// TwinCAT 3 PLC project PLC
// ProgramVersion: 3.1.4023.0
// libraries:
//   Tc2_Standard, * (Beckhoff Automation GmbH)
//   Tc2_System, * (Beckhoff Automation GmbH)
//   Tc3_Module, * (Beckhoff Automation GmbH)
// project tree:
//   / PlcTask.TcTTO
//   POUs/ MAIN.TcPOU
//   DUTs/IO/PDOs/ InfoData_6F19DB2B.TcDUT, Inputs_CC16D1F4.TcDUT, Outputs_D8BAB3B3.TcDUT, WcState_9091E0EB.TcDUT, InfoData_90184F0C.TcDUT, Channel_87C95E76.TcDUT, InfoData_32EB74EA.TcDUT, Channel_70C997F3.TcDUT, EPM_Inputs_Channel_385E794A.TcDUT, EMPTY_STRUCTURE.TcDUT, Device_Status_Mapping_61F79077.TcDUT, Channel_954C2EED.TcDUT, Channel_60E28ED2.TcDUT, Channel_7DE26195.TcDUT, Channel_2E0D480D.TcDUT, Channel_61FC1536.TcDUT, Channel_16463F74.TcDUT, Channel_707BD1FE.TcDUT, Channel_7D202F58.TcDUT, Channel_6CC0E226.TcDUT, Channel_0F0CD940.TcDUT, Channel_65B76600.TcDUT, Channel_72DF6336.TcDUT, Channel_22DCD695.TcDUT, Channel_3C1A6500.TcDUT, Channel_B5275D8E.TcDUT, Channel_03CEAA5E.TcDUT, Channel_1D6668A9.TcDUT, Channel_6B723A16.TcDUT, Channel_460B8C40.TcDUT, Channel_DCF170BB.TcDUT, Channel_26FC8FD8.TcDUT, Channel_FEA3DBF8.TcDUT, Channel_0D1929F0.TcDUT, Channel_6576A681.TcDUT, Channel_2589C8DC.TcDUT, Channel_BF3661CD.TcDUT, Channel_2EC3E8CA.TcDUT, Channel_F5DB8AD1.TcDUT, Channel_6D8B740B.TcDUT, Channel_2DA3FF3C.TcDUT, Channel_0514A8FA.TcDUT, Channel_4E9D1E2D.TcDUT, Channel_78571FB4.TcDUT, Channel_87905831.TcDUT, Channel_099BCCDA.TcDUT, Channel_82ADD076.TcDUT, Channel_332F026B.TcDUT, Channel_A6A8AB45.TcDUT, Channel_A42BCA5C.TcDUT, Channel_08506BCE.TcDUT, Channel_08533804.TcDUT, Channel_A04AC4BD.TcDUT, Channel_77910383.TcDUT, Channel_9BC0092E.TcDUT, Channel_7606D989.TcDUT, Channel_6931CC5B.TcDUT, Channel_F7FDEFA0.TcDUT, Channel_A1C14FB4.TcDUT, Channel_A4B48F2D.TcDUT, Channel_9E293686.TcDUT, Channel_F84AC14F.TcDUT, Channel_2F314509.TcDUT, Channel_D9D48807.TcDUT, Channel_D13646E3.TcDUT, Channel_3263D8D5.TcDUT, Channel_D490E973.TcDUT, KL_6576A681.TcDUT, Channel_64AAC8C7.TcDUT, Channel_471FAA5C.TcDUT, Diag_1F4F4573.TcDUT, Channel_0029832E.TcDUT, Channel_12652743.TcDUT, InfoData_E68C61CD.TcDUT, WcState_0B2B16F9.TcDUT, InfoData_2A97D6CF.TcDUT, Inputs_25A0042B.TcDUT, Outputs_2397A10E.TcDUT
//   DUTs/IO/Boxes/ EK1100_1FC0878B.TcDUT, EK1122_1FC0878B.TcDUT, BK1250_A2FCADE7.TcDUT, KL1002_BB38DA8F.TcDUT, BK1120_6D44499E.TcDUT, BK1120_A2FCADE7.TcDUT, CPXXXX_A2FCADE7.TcDUT, BK1150_A2FCADE7.TcDUT, IL2300_A2FCADE7.TcDUT, KL_D4CFBC22.TcDUT, KL_8EF4D3E9.TcDUT, IL2301_A2FCADE7.TcDUT, IL2302_A2FCADE7.TcDUT, CU1123_1FC0878B.TcDUT, CU1124_1FC0878B.TcDUT, CU1128_1FC0878B.TcDUT, CU1521_1FC0878B.TcDUT, CU1561_1FC0878B.TcDUT, CU2508_1FC0878B.TcDUT, CU2508_EEB2FEF4.TcDUT, CU2508_6BF2ACBC.TcDUT, CX1100_1FC0878B.TcDUT, CX5010_EtherCAT_slave_FEF7A27A.TcDUT, CX5020_EtherCAT_slave_FEF7A27A.TcDUT, CX8010_EtherCAT_slave_FEF7A27A.TcDUT, CX8110_EtherCAT_slave_FEF7A27A.TcDUT, CX2020_EtherCAT_slave_FEF7A27A.TcDUT, CX2030_EtherCAT_slave_FEF7A27A.TcDUT, CX2033_EtherCAT_slave_FEF7A27A.TcDUT, CX2040_EtherCAT_slave_FEF7A27A.TcDUT, CX2042_EtherCAT_slave_FEF7A27A.TcDUT, CX2043_EtherCAT_slave_FEF7A27A.TcDUT, CX2062_EtherCAT_slave_FEF7A27A.TcDUT, CX2072_EtherCAT_slave_FEF7A27A.TcDUT, CX9020_EtherCAT_slave_FEF7A27A.TcDUT, CX5120_EtherCAT_slave_FEF7A27A.TcDUT, CX5130_EtherCAT_slave_FEF7A27A.TcDUT, CX5140_EtherCAT_slave_FEF7A27A.TcDUT, CX5230_EtherCAT_slave_FEF7A27A.TcDUT, CX5240_EtherCAT_slave_FEF7A27A.TcDUT, KL_5E2F016F.TcDUT, KL_2EA97E3E.TcDUT, KL_1187B721.TcDUT, KL_E991A364.TcDUT, KL_063F0990.TcDUT, KL_5AE00A1C.TcDUT, KL_CFA8830D.TcDUT, KL_DBC0B844.TcDUT, KL_6930B3B2.TcDUT, KL_4F0DAD84.TcDUT, KL_2227C35B.TcDUT, KL_E653A8C1.TcDUT, KL1012_BB38DA8F.TcDUT, KL1032_BB38DA8F.TcDUT, KL1052_BB38DA8F.TcDUT, KL1104_4A257D2B.TcDUT, KL1114_4A257D2B.TcDUT, KL1124_4A257D2B.TcDUT, KL1154_4A257D2B.TcDUT, KL1164_4A257D2B.TcDUT, KL1184_4A257D2B.TcDUT, KL1194_4A257D2B.TcDUT, KL1212_EC84F46C.TcDUT, KL1232_BB38DA8F.TcDUT, KL1302_BB38DA8F.TcDUT, KL1304_4A257D2B.TcDUT, KL1312_BB38DA8F.TcDUT, KL1314_4A257D2B.TcDUT, KL1352_B54AC54D.TcDUT, KL1362_B54AC54D.TcDUT, KL1382_B54AC54D.TcDUT, KL1402_BB38DA8F.TcDUT, KL1404_4A257D2B.TcDUT, KL1408_8EF4D3E9.TcDUT, KL1412_BB38DA8F.TcDUT, KL1414_4A257D2B.TcDUT, KL1418_8EF4D3E9.TcDUT, KL1434_4A257D2B.TcDUT, KL1488_8EF4D3E9.TcDUT, KL1498_8EF4D3E9.TcDUT, KL1501_EE1D4506.TcDUT, KL_62DC61BC.TcDUT, KL1512_78388DBB.TcDUT, KL1702_BB38DA8F.TcDUT, KL1704_4A257D2B.TcDUT, KL1712_BB38DA8F.TcDUT, KL_BB38DA8F.TcDUT, KL1722_BB38DA8F.TcDUT, KL1804_4A257D2B.TcDUT, KL1808_8EF4D3E9.TcDUT, KL1809_65B88BEE.TcDUT, KL1814_4A257D2B.TcDUT, KL1819_65B88BEE.TcDUT, KL1859_C5B2A062.TcDUT, KL1862_65B88BEE.TcDUT, KL_65B88BEE.TcDUT, KL1872_65B88BEE.TcDUT, KL1889_65B88BEE.TcDUT, KL1904_7F0D69A9.TcDUT, KL1908_7F0D69A9.TcDUT, KL_ABE34026.TcDUT, KL_E882B8F1.TcDUT, KL_52751275.TcDUT, KL2012_DCA75612.TcDUT, KL2022_DCA75612.TcDUT, KL2032_DCA75612.TcDUT, KL2114_E49EE1EF.TcDUT, KL2124_E49EE1EF.TcDUT, KL2134_E49EE1EF.TcDUT, KL2184_E49EE1EF.TcDUT, KL2212_BA18203A.TcDUT, KL1202_EC84F46C.TcDUT, KL2404_E49EE1EF.TcDUT, KL2408_CBAD53BF.TcDUT, KL2424_E49EE1EF.TcDUT, KL2442_DCA75612.TcDUT, KL2488_CBAD53BF.TcDUT, KL2284_008A18FD.TcDUT, KL2502_78388DBB.TcDUT, KL2512_78388DBB.TcDUT, KL2521_D5F34107.TcDUT, KL2531_D5AE5504.TcDUT, KL_5C335388.TcDUT, KL2532_B0461874.TcDUT, KL2535_B0461874.TcDUT, KL_501418F2.TcDUT, KL2541_D5AE5504.TcDUT, KL2542_B0461874.TcDUT, KL2545_B0461874.TcDUT, KL2552_B0461874.TcDUT, KL2602_DCA75612.TcDUT, KL_DCA75612.TcDUT, KL2612_DCA75612.TcDUT, KL2622_DCA75612.TcDUT, KL2631_DE78D366.TcDUT, KL2634_E49EE1EF.TcDUT, KL2641_8487B205.TcDUT, KL_AF699C3C.TcDUT, KL2652_DCA75612.TcDUT, KL_6148C904.TcDUT, KL2701_DE78D366.TcDUT, KL2702_DCA75612.TcDUT, KL2712_DCA75612.TcDUT, KL2722_DCA75612.TcDUT, KL2732_DCA75612.TcDUT, KL2744_E49EE1EF.TcDUT, KL2751_6148C904.TcDUT, KL2761_6148C904.TcDUT, KL2784_E49EE1EF.TcDUT, KL2791_6148C904.TcDUT, KL2794_E49EE1EF.TcDUT, KL2798_CBAD53BF.TcDUT, KL2808_CBAD53BF.TcDUT, KL2819_28D63841.TcDUT, KL2828_CBAD53BF.TcDUT, KL2809_F0D0C9F8.TcDUT, KL2872_F0D0C9F8.TcDUT, KL2889_F0D0C9F8.TcDUT, KL2904_7F0D69A9.TcDUT, KL_F0D0C9F8.TcDUT, KL_CF002DCA.TcDUT, KL_F7A5EEBF.TcDUT, KL_E49EE1EF.TcDUT, KL_F206FFFF.TcDUT, KL_13ED1AE5.TcDUT, KL2774_6148C904.TcDUT, KL_CBAD53BF.TcDUT, KL3001_6148C904.TcDUT, KL3002_B0461874.TcDUT, KL3011_6148C904.TcDUT, KL3012_B0461874.TcDUT, KL3021_6148C904.TcDUT, KL3022_B0461874.TcDUT, KL3041_6148C904.TcDUT, KL3042_B0461874.TcDUT, KL3044_8BE38B75.TcDUT, KL_ACD69469.TcDUT, KL3051_6148C904.TcDUT, KL3052_B0461874.TcDUT, KL3054_8BE38B75.TcDUT, KL3061_6148C904.TcDUT, KL3062_B0461874.TcDUT, KL3064_8BE38B75.TcDUT, KL3102_B0461874.TcDUT, KL3112_B0461874.TcDUT, KL3122_B0461874.TcDUT, KL3132_B0461874.TcDUT, KL3142_78388DBB.TcDUT, KL3152_78388DBB.TcDUT, KL3158_8BE38B75.TcDUT, KL3162_78388DBB.TcDUT, KL3172_78388DBB.TcDUT, KL_78388DBB.TcDUT, KL3182_B0461874.TcDUT, KL3201_6148C904.TcDUT, KL3202_B0461874.TcDUT, KL3204_8BE38B75.TcDUT, KL_8BE38B75.TcDUT, KL3214_8BE38B75.TcDUT, KL3222_B0461874.TcDUT, KL3224_8BE38B75.TcDUT, KL3228_8BE38B75.TcDUT, KL3302_B0461874.TcDUT, KL3311_6148C904.TcDUT, KL3312_B0461874.TcDUT, KL3314_8BE38B75.TcDUT, KL3351_33637CB0.TcDUT, KL_C7B8B3CA.TcDUT, KL3356_E004D4E2.TcDUT, KL_EE1D4506.TcDUT, KL3361_73CB82BA.TcDUT, KL_73CB82BA.TcDUT, KL3362_E98BF8F1.TcDUT, KL6211_60136EA1.TcDUT, KL_9AE543B6.TcDUT, KL_FC0201B8.TcDUT, KL_498D8863.TcDUT, KL_71341691.TcDUT, KL_2B11657C.TcDUT, KL6224_C0F107BD.TcDUT, KL_FC1E3393.TcDUT, KL_C51B1CB0.TcDUT, KL_7EC2CD64.TcDUT, KL_3829421A.TcDUT, KL_9116C2C1.TcDUT, KL6551_528AE398.TcDUT, KL_3325E583.TcDUT, KL_528AE398.TcDUT, KL6781_BE595CA2.TcDUT, KL6811_6148C904.TcDUT, KL6821_F77C82D2.TcDUT, KL6831_BE595CA2.TcDUT, KL6841_BE595CA2.TcDUT, KL6904_B938D612.TcDUT, KL_921B772D.TcDUT, KL_779990DF.TcDUT, KL8001_7761653A.TcDUT, KL8519_8C34650F.TcDUT, KL8524_A4B9216E.TcDUT, KL8528_73A97EC1.TcDUT, KL8548_23451728.TcDUT, KL8610_C571D068.TcDUT, KL_5A83E84C.TcDUT, KL_BF4AA06C.TcDUT, KL_7485E925.TcDUT, KL_372C6BEC.TcDUT, KL_2E5CD6C8.TcDUT, KL_68BDE1E9.TcDUT, KL_84AAE8B6.TcDUT, KL9110_8BEE55F2.TcDUT, KL9160_8BEE55F2.TcDUT, KL9191_962A24DF.TcDUT, KL9210_8BEE55F2.TcDUT, KL9260_8BEE55F2.TcDUT, KL_E4BD2B38.TcDUT, KL9528_8C984603.TcDUT, KL9999_7A10A7F6.TcDUT
//   DUTs/IO/Devices/ SyncUnitTask_2D604ED5.TcDUT, SyncUnitTasks_6FEB8257.TcDUT, SyncUnits_99E584AF.TcDUT
//   DUTs/IO/Topology/ A_0014_BK1250_0000_0000_09E1EB45.TcDUT, Beckhoff_BKxxxxsub_EK1100_59A46924.TcDUT, A_0001_BK1120_0000_0000_205E6559.TcDUT, A_0002_BK1120_0000_0001_76F1F8EB.TcDUT, A_0003_BK1120_0000_0016_8D015E3D.TcDUT, A_0004_BK1120_0000_0017_DBAEC38F.TcDUT, A_0005_BK1120_0000_0018_C2DFD8D8.TcDUT, A_0006_BK1120_0000_0019_9470456A.TcDUT, A_0007_BK1120_0000_0020_61E27259.TcDUT, A_0008_BK1120_0000_0021_374DEFEB.TcDUT, A_0009_CPXXXX_BK1150_0016_CCBD493D.TcDUT, A_0010_BK1150_0000_0016_9A12D48F.TcDUT, A_0011_BK1150_0000_0017_3F9D1926.TcDUT, A_0012_BK1150_0000_0018_69328494.TcDUT, A_0013_BK1150_0000_0019_92C22242.TcDUT, A_0016_BK1250_0000_0017_C46DBFF0.TcDUT, Term_19_EK1100_718FBBA4.TcDUT, A_0018_BK1250_0000_0019_DD1CA4A7.TcDUT, Term_23_EK1100_08A82DAA.TcDUT, A_0017_BK1250_0000_0018_8BB33915.TcDUT, Term_21_EK1100_FD75FF18.TcDUT, A_0019_IL2300_B110_0016_AC908CDE.TcDUT, A_0020_IL2300_B110_0017_8C062E24.TcDUT, A_0021_IL2301_B110_0016_FF61810D.TcDUT, A_0022_IL2301_B110_0017_BAC34F2E.TcDUT, A_0023_IL2302_B110_0016_19AEDF5F.TcDUT, A_0024_IL2302_B110_0017_E18CEC30.TcDUT, Beckhoff_BKxxxxEK1122_C32C6A5C.TcDUT, A_0015_BK1250_0000_0016_5F4E76F7.TcDUT, Beckhoff_BKxxxx_735133AB.TcDUT, A_0006_CU1128_0000_0002_093CCA2E.TcDUT, A_0005_CU1128_0000_0001_8DEFD527.TcDUT, A_0004_CU1128_0000_0000_2F60DA9F.TcDUT, A_0003_CU1124_0000_0016_CE6B0448.TcDUT, A_0002_CU1123_0010_0016_E68B3D99.TcDUT, A_0001_CU1123_0000_0016_30E128CC.TcDUT, Beckhoff_CUxxxxEK1122_BE344318.TcDUT, Beckhoff_CUxxxx_E9AD9532.TcDUT, Beckhoff_CXxxxxEK1122_ADC91C0D.TcDUT, Beckhoff_CXxxxx_7C0A3C1E.TcDUT, TcTerminals210_1BK1250_A7ABB5AA.TcDUT, TcTerminals210_EK1100_1_5C778379.TcDUT, TcTerminals210_2BK1250_CEF74155.TcDUT, TcTerminals210_EK1100_2_50C14331.TcDUT, EtherCAT_Master_BKCUCX_25A199DC.TcDUT
//   DUTs/IO/Base/ EtcSlaveBase_82538BE2.TcDUT, EtcSlaveBase_82538BE2.TcDUT, EtcSlaveBase_82538BE2.TcDUT, EtcSlaveTerminalBase_947E5A46.TcDUT, EtcSlaveBoxBase_77A0E4A7.TcDUT, EtcSlaveEndTerminalBase_866C7F0C.TcDUT, InputBase_8311D824.TcDUT, OutputBase_10CEE7DE.TcDUT, EtcMasterBase_62654B43.TcDUT
//   GVLs/ GVL_iXlinker.TcGVL
// real-time tasks:
//   TASK PlcTask: cycle T#10ms, priority 20, ADS port 350
// I/O:
//   DEVICE EtherCAT_Master_BKCUCX, AmsNetId 172.20.30.238.6.1
//     Beckhoff BKxxxx [EK1100 EtherCAT Coupler (2A E-Bus)]
//       Beckhoff BKxxxxEK1122 [EK1122 2 port EtherCAT junction]
//         Beckhoff BKxxxxsub EK1100 [EK1100 EtherCAT Coupler (2A E-Bus)]
//           A_0014(BK1250-0000-0000)
//         A_0001(BK1120-0000-0000)
//         A_0002(BK1120-0000-0001)
//         A_0003(BK1120-0000-0016)
//         A_0004(BK1120-0000-0017)
//         A_0005(BK1120-0000-0018)
//         A_0006(BK1120-0000-0019)
//         A_0007(BK1120-0000-0020)
//         A_0008(BK1120-0000-0021)
//         A_0009(CPXXXX-BK1150-0016)
//         A_0010(BK1150-0000-0016)
//         A_0011(BK1150-0000-0017)
//         A_0012(BK1150-0000-0018)
//         A_0013(BK1150-0000-0019)
//         Term 19 (EK1100) [EK1100 EtherCAT Coupler (2A E-Bus)]
//           A_0016(BK1250-0000-0017)
//         Term 23 (EK1100) [EK1100 EtherCAT Coupler (2A E-Bus)]
//           A_0018(BK1250-0000-0019)
//         Term 21 (EK1100) [EK1100 EtherCAT Coupler (2A E-Bus)]
//           A_0017(BK1250-0000-0018)
//         A_0019(IL2300-B110-0016)
//         A_0020(IL2300-B110-0017)
//         A_0021(IL2301-B110-0016)
//         A_0022(IL2301-B110-0017)
//         A_0023(IL2302-B110-0016)
//         A_0024(IL2302-B110-0017)
//       A_0015(BK1250-0000-0016)
//     Beckhoff CUxxxx [EK1100 EtherCAT Coupler (2A E-Bus)]
//       Beckhoff CUxxxxEK1122 [EK1122 2 port EtherCAT junction]
//         Beckhoff CUxxxxsub EK1100 [EK1100 EtherCAT Coupler (2A E-Bus)]
//         A_0001(CU1123-0000-0016) [CU1123 EtherCAT junction (3-ports)]
//           A_0002(CU1123-0010-0016) [CU1123-0010 EtherCAT junction (3-ports, Extended Distance)]
//             A_0003(CU1124-0000-0016) [CU1124 EtherCAT junction (4-ports)]
//               A_0004(CU1128-0000-0000) [CU1128 6x EtherCAT junction]
//                 A_0005(CU1128-0000-0001) [CU1128 6x EtherCAT junction]
//                   A_0006(CU1128-0000-0002) [CU1128 6x EtherCAT junction]
//                     A_0007(CU1521-0010-0000) [CU1521-0010 EtherCAT media converter (Singlemode)]
//                     A_0008(CU1561-0000-0000) [CU1561 EtherCAT media converter (POF)]
//                     A_0009(CU2508-0000-0000) [CU2508 Ethernet Port]
//                     A_0010(CU2508-0000-0016) [CU2508 Configuration Port]
//                     A_0011(CU2508-0000-0017) [CU2508 Configuration Port]
//                     A_0012(CU2508-0000-0018) [CU2508 Configuration Port]
//                     A_0013(CU2508-0000-0019) [CU2508 Configuration Port]
//                     A_0006(CU1128-0000-0002)_2 (CU1128-B) [CU1128 6x EtherCAT junction - Dev A]
//                     A_0006(CU1128-0000-0002)_3 (CU1128-C) [CU1128 6x EtherCAT junction - Dev B]
//                   A_0005(CU1128-0000-0001)_2 (CU1128-B) [CU1128 6x EtherCAT junction - Dev A]
//                   A_0005(CU1128-0000-0001)_3 (CU1128-C) [CU1128 6x EtherCAT junction - Dev B]
//                 A_0004(CU1128-0000-0000)_2 (CU1128-B) [CU1128 6x EtherCAT junction - Dev A]
//                 A_0004(CU1128-0000-0000)_3 (CU1128-C) [CU1128 6x EtherCAT junction - Dev B]
//     Beckhoff CXxxxx [EK1100 EtherCAT Coupler (2A E-Bus)]
//       Beckhoff CXxxxxEK1122 [EK1122 2 port EtherCAT junction]
//         Beckhoff CXxxxxsub EK1100 [EK1100 EtherCAT Coupler (2A E-Bus)]
//         A_0001(CX1100-0004-0000) [CX1100-0004 EtherCAT Power supply (2A E-Bus)]
//         A_0003(CX1100-0004-0002) [CX1100-0004 EtherCAT Power supply (2A E-Bus)]
//         A_0004 (CX5010 EtherCAT slave) [CX5010 EtherCAT slave]
//         A_0005 (CX5010 EtherCAT slave) [CX5010 EtherCAT slave]
//         A_0006 (CX5020 EtherCAT slave) [CX5020 EtherCAT slave]
//         A_0007 (CX5020 EtherCAT slave) [CX5020 EtherCAT slave]
//         A_0008 (CX8010 EtherCAT slave) [CX8010 EtherCAT slave]
//         A_0009 (CX8010 EtherCAT slave) [CX8010 EtherCAT slave]
//         A_0010 (CX8110 EtherCAT slave) [CX8110 EtherCAT slave]
//         A_0011 (CX2020 EtherCAT slave) [CX2020 EtherCAT slave]
//         A_0012 (CX2020 EtherCAT slave) [CX2020 EtherCAT slave]
//         A_0013 (CX2020 EtherCAT slave) [CX2020 EtherCAT slave]
//         A_0014 (CX2030 EtherCAT slave) [CX2030 EtherCAT slave]
//         A_0015 (CX2030 EtherCAT slave) [CX2030 EtherCAT slave]
//         A_0016 (CX2030 EtherCAT slave) [CX2030 EtherCAT slave]
//         A_0017 (CX2033 EtherCAT slave) [CX2033 EtherCAT slave]
//         A_0018 (CX2040 EtherCAT slave) [CX2040 EtherCAT slave]
//         A_0019 (CX2040 EtherCAT slave) [CX2040 EtherCAT slave]
//         A_0020 (CX2040 EtherCAT slave) [CX2040 EtherCAT slave]
//         A_0021 (CX2042 EtherCAT slave) [CX2042 EtherCAT slave]
//         A_0022 (CX2043 EtherCAT slave) [CX2043 EtherCAT slave]
//         A_0023 (CX2062 EtherCAT slave) [CX2062 EtherCAT slave]
//         A_0024 (CX2072 EtherCAT slave) [CX2072 EtherCAT slave]
//         A_0025 (CX9020 EtherCAT slave) [CX9020 EtherCAT slave]
//         A_0026 (CX9020 EtherCAT slave) [CX9020 EtherCAT slave]
//         A_0027 (CX5120 EtherCAT slave) [CX5120 EtherCAT slave]
//         A_0028 (CX5130 EtherCAT slave) [CX5130 EtherCAT slave]
//         A_0029 (CX5140 EtherCAT slave) [CX5140 EtherCAT slave]
//         A_0030 (CX5230 EtherCAT slave) [CX5230 EtherCAT slave]
//         A_0031 (CX5240 EtherCAT slave) [CX5240 EtherCAT slave]
//         A_0002(CX1100-0004-0001) [CX1100-0004 EtherCAT Power supply (2A E-Bus)]
//     TcTerminals210_EK1100_1 [EK1100 EtherCAT Coupler (2A E-Bus)]
//       TcTerminals210_1BK1250
//     TcTerminals210_EK1100_2 [EK1100 EtherCAT Coupler (2A E-Bus)]
//       TcTerminals210_2BK1250
// variable links:
//   PLC/PLC Instance <-> EtherCAT Master BKCUCX/Beckhoff BKxxxx
//     PlcTask Inputs/GVL_iXlinker.EtherCAT_Master_BKCUCX.Beckhoff_BKxxxx.InfoData.State <-> InfoData/State
//   PLC/PLC Instance <-> EtherCAT Master BKCUCX/Beckhoff BKxxxx/Beckhoff BKxxxxEK1122
//     PlcTask Inputs/GVL_iXlinker.EtherCAT_Master_BKCUCX.Beckhoff_BKxxxx.Beckhoff_BKxxxxEK1122.InfoData.State <-> InfoData/State
//   PLC/PLC Instance <-> EtherCAT Master BKCUCX/Beckhoff BKxxxx/Beckhoff BKxxxxEK1122/Beckhoff BKxxxxsub EK1100
//     PlcTask Inputs/GVL_iXlinker.EtherCAT_Master_BKCUCX.Beckhoff_BKxxxx.Beckhoff_BKxxxxEK1122.Beckhoff_BKxxxxsub_EK1100.InfoData.State <-> InfoData/State
//   PLC/PLC Instance <-> EtherCAT Master BKCUCX/Beckhoff BKxxxx/Beckhoff BKxxxxEK1122/Beckhoff BKxxxxsub EK1100/A_0014(BK1250-0000-0000)
//     PlcTask Inputs/GVL_iXlinker.EtherCAT_Master_BKCUCX.Beckhoff_BKxxxx.Beckhoff_BKxxxxEK1122.Beckhoff_BKxxxxsub_EK1100.A_0014_BK1250_0000_0000.Inputs.CouplerState <-> Inputs/CouplerState
//     PlcTask Inputs/GVL_iXlinker.EtherCAT_Master_BKCUCX.Beckhoff_BKxxxx.Beckhoff_BKxxxxEK1122.Beckhoff_BKxxxxsub_EK1100.A_0014_BK1250_0000_0000.Outputs.CouplerCtrl <-> Outputs/CouplerCtrl
//     PlcTask Inputs/GVL_iXlinker.EtherCAT_Master_BKCUCX.Beckhoff_BKxxxx.Beckhoff_BKxxxxEK1122.Beckhoff_BKxxxxsub_EK1100.A_0014_BK1250_0000_0000.WcState.WcState <-> WcState/WcState
//     PlcTask Inputs/GVL_iXlinker.EtherCAT_Master_BKCUCX.Beckhoff_BKxxxx.Beckhoff_BKxxxxEK1122.Beckhoff_BKxxxxsub_EK1100.A_0014_BK1250_0000_0000.WcState.InputToggle <-> WcState/InputToggle
//     PlcTask Inputs/GVL_iXlinker.EtherCAT_Master_BKCUCX.Beckhoff_BKxxxx.Beckhoff_BKxxxxEK1122.Beckhoff_BKxxxxsub_EK1100.A_0014_BK1250_0000_0000.InfoData.AdsAddr <-> InfoData/AdsAddr
//     PlcTask Inputs/GVL_iXlinker.EtherCAT_Master_BKCUCX.Beckhoff_BKxxxx.Beckhoff_BKxxxxEK1122.Beckhoff_BKxxxxsub_EK1100.A_0014_BK1250_0000_0000.InfoData.AoeNetId <-> InfoData/AoeNetId
//     PlcTask Inputs/GVL_iXlinker.EtherCAT_Master_BKCUCX.Beckhoff_BKxxxx.Beckhoff_BKxxxxEK1122.Beckhoff_BKxxxxsub_EK1100.A_0014_BK1250_0000_0000.InfoData.State <-> InfoData/State
//   PLC/PLC Instance <-> EtherCAT Master BKCUCX/Beckhoff BKxxxx/Beckhoff BKxxxxEK1122/Beckhoff BKxxxxsub EK1100/A_0014(BK1250-0000-0000)/Term 397 (KL1002)
//     PlcTask Inputs/GVL_iXlinker.EtherCAT_Master_BKCUCX.Beckhoff_BKxxxx.Beckhoff_BKxxxxEK1122.Beckhoff_BKxxxxsub_EK1100.A_0014_BK1250_0000_0000.Term_397_KL1002.Channel_1.Input <-> Channel 1/Input
//     PlcTask Inputs/GVL_iXlinker.EtherCAT_Master_BKCUCX.Beckhoff_BKxxxx.Beckhoff_BKxxxxEK1122.Beckhoff_BKxxxxsub_EK1100.A_0014_BK1250_0000_0000.Term_397_KL1002.Channel_2.Input <-> Channel 2/Input
//   PLC/PLC Instance <-> EtherCAT Master BKCUCX/Beckhoff BKxxxx/Beckhoff BKxxxxEK1122/A_0001(BK1120-0000-0000)
//     PlcTask Inputs/GVL_iXlinker.EtherCAT_Master_BKCUCX.Beckhoff_BKxxxx.Beckhoff_BKxxxxEK1122.A_0001_BK1120_0000_0000.Inputs.CouplerState <-> Inputs/CouplerState
//     PlcTask Inputs/GVL_iXlinker.EtherCAT_Master_BKCUCX.Beckhoff_BKxxxx.Beckhoff_BKxxxxEK1122.A_0001_BK1120_0000_0000.Outputs.CouplerCtrl <-> Outputs/CouplerCtrl
//     PlcTask Inputs/GVL_iXlinker.EtherCAT_Master_BKCUCX.Beckhoff_BKxxxx.Beckhoff_BKxxxxEK1122.A_0001_BK1120_0000_0000.WcState.WcState <-> WcState/WcState
//     PlcTask Inputs/GVL_iXlinker.EtherCAT_Master_BKCUCX.Beckhoff_BKxxxx.Beckhoff_BKxxxxEK1122.A_0001_BK1120_0000_0000.WcState.InputToggle <-> WcState/InputToggle
//     PlcTask Inputs/GVL_iXlinker.EtherCAT_Master_BKCUCX.Beckhoff_BKxxxx.Beckhoff_BKxxxxEK1122.A_0001_BK1120_0000_0000.InfoData.AdsAddr <-> InfoData/AdsAddr
//     PlcTask Inputs/GVL_iXlinker.EtherCAT_Master_BKCUCX.Beckhoff_BKxxxx.Beckhoff_BKxxxxEK1122.A_0001_BK1120_0000_0000.InfoData.State <-> InfoData/State
//   PLC/PLC Instance <-> EtherCAT Master BKCUCX/Beckhoff BKxxxx/Beckhoff BKxxxxEK1122/A_0001(BK1120-0000-0000)/Term 374 (KL1002)
//     PlcTask Inputs/GVL_iXlinker.EtherCAT_Master_BKCUCX.Beckhoff_BKxxxx.Beckhoff_BKxxxxEK1122.A_0001_BK1120_0000_0000.Term_374_KL1002.Channel_1.Input <-> Channel 1/Input
//     PlcTask Inputs/GVL_iXlinker.EtherCAT_Master_BKCUCX.Beckhoff_BKxxxx.Beckhoff_BKxxxxEK1122.A_0001_BK1120_0000_0000.Term_374_KL1002.Channel_2.Input <-> Channel 2/Input
//   PLC/PLC Instance <-> EtherCAT Master BKCUCX/Beckhoff BKxxxx/Beckhoff BKxxxxEK1122/A_0002(BK1120-0000-0001)
//     PlcTask Inputs/GVL_iXlinker.EtherCAT_Master_BKCUCX.Beckhoff_BKxxxx.Beckhoff_BKxxxxEK1122.A_0002_BK1120_0000_0001.Inputs.CouplerState <-> Inputs/CouplerState
//     PlcTask Inputs/GVL_iXlinker.EtherCAT_Master_BKCUCX.Beckhoff_BKxxxx.Beckhoff_BKxxxxEK1122.A_0002_BK1120_0000_0001.Outputs.CouplerCtrl <-> Outputs/CouplerCtrl
//     PlcTask Inputs/GVL_iXlinker.EtherCAT_Master_BKCUCX.Beckhoff_BKxxxx.Beckhoff_BKxxxxEK1122.A_0002_BK1120_0000_0001.WcState.WcState <-> WcState/WcState
//     PlcTask Inputs/GVL_iXlinker.EtherCAT_Master_BKCUCX.Beckhoff_BKxxxx.Beckhoff_BKxxxxEK1122.A_0002_BK1120_0000_0001.WcState.InputToggle <-> WcState/InputToggle
//     PlcTask Inputs/GVL_iXlinker.EtherCAT_Master_BKCUCX.Beckhoff_BKxxxx.Beckhoff_BKxxxxEK1122.A_0002_BK1120_0000_0001.InfoData.AdsAddr <-> InfoData/AdsAddr
//     PlcTask Inputs/GVL_iXlinker.EtherCAT_Master_BKCUCX.Beckhoff_BKxxxx.Beckhoff_BKxxxxEK1122.A_0002_BK1120_0000_0001.InfoData.AoeNetId <-> InfoData/AoeNetId
//     PlcTask Inputs/GVL_iXlinker.EtherCAT_Master_BKCUCX.Beckhoff_BKxxxx.Beckhoff_BKxxxxEK1122.A_0002_BK1120_0000_0001.InfoData.State <-> InfoData/State
//   PLC/PLC Instance <-> EtherCAT Master BKCUCX/Beckhoff BKxxxx/Beckhoff BKxxxxEK1122/A_0002(BK1120-0000-0001)/Term 375 (KL1002)
//     PlcTask Inputs/GVL_iXlinker.EtherCAT_Master_BKCUCX.Beckhoff_BKxxxx.Beckhoff_BKxxxxEK1122.A_0002_BK1120_0000_0001.Term_375_KL1002.Channel_1.Input <-> Channel 1/Input
//     PlcTask Inputs/GVL_iXlinker.EtherCAT_Master_BKCUCX.Beckhoff_BKxxxx.Beckhoff_BKxxxxEK1122.A_0002_BK1120_0000_0001.Term_375_KL1002.Channel_2.Input <-> Channel 2/Input
//   PLC/PLC Instance <-> EtherCAT Master BKCUCX/Beckhoff BKxxxx/Beckhoff BKxxxxEK1122/A_0003(BK1120-0000-0016)
//     PlcTask Inputs/GVL_iXlinker.EtherCAT_Master_BKCUCX.Beckhoff_BKxxxx.Beckhoff_BKxxxxEK1122.A_0003_BK1120_0000_0016.Inputs.CouplerState <-> Inputs/CouplerState
//     PlcTask Inputs/GVL_iXlinker.EtherCAT_Master_BKCUCX.Beckhoff_BKxxxx.Beckhoff_BKxxxxEK1122.A_0003_BK1120_0000_0016.Outputs.CouplerCtrl <-> Outputs/CouplerCtrl
//     PlcTask Inputs/GVL_iXlinker.EtherCAT_Master_BKCUCX.Beckhoff_BKxxxx.Beckhoff_BKxxxxEK1122.A_0003_BK1120_0000_0016.WcState.WcState <-> WcState/WcState
//     PlcTask Inputs/GVL_iXlinker.EtherCAT_Master_BKCUCX.Beckhoff_BKxxxx.Beckhoff_BKxxxxEK1122.A_0003_BK1120_0000_0016.WcState.InputToggle <-> WcState/InputToggle
//     PlcTask Inputs/GVL_iXlinker.EtherCAT_Master_BKCUCX.Beckhoff_BKxxxx.Beckhoff_BKxxxxEK1122.A_0003_BK1120_0000_0016.InfoData.AdsAddr <-> InfoData/AdsAddr
//     PlcTask Inputs/GVL_iXlinker.EtherCAT_Master_BKCUCX.Beckhoff_BKxxxx.Beckhoff_BKxxxxEK1122.A_0003_BK1120_0000_0016.InfoData.AoeNetId <-> InfoData/AoeNetId
//     PlcTask Inputs/GVL_iXlinker.EtherCAT_Master_BKCUCX.Beckhoff_BKxxxx.Beckhoff_BKxxxxEK1122.A_0003_BK1120_0000_0016.InfoData.State <-> InfoData/State
//   PLC/PLC Instance <-> EtherCAT Master BKCUCX/Beckhoff BKxxxx/Beckhoff BKxxxxEK1122/A_0003(BK1120-0000-0016)/Term 376 (KL1002)
//     PlcTask Inputs/GVL_iXlinker.EtherCAT_Master_BKCUCX.Beckhoff_BKxxxx.Beckhoff_BKxxxxEK1122.A_0003_BK1120_0000_0016.Term_376_KL1002.Channel_1.Input <-> Channel 1/Input
//     PlcTask Inputs/GVL_iXlinker.EtherCAT_Master_BKCUCX.Beckhoff_BKxxxx.Beckhoff_BKxxxxEK1122.A_0003_BK1120_0000_0016.Term_376_KL1002.Channel_2.Input <-> Channel 2/Input
//   PLC/PLC Instance <-> EtherCAT Master BKCUCX/Beckhoff BKxxxx/Beckhoff BKxxxxEK1122/A_0004(BK1120-0000-0017)
//     PlcTask Inputs/GVL_iXlinker.EtherCAT_Master_BKCUCX.Beckhoff_BKxxxx.Beckhoff_BKxxxxEK1122.A_0004_BK1120_0000_0017.Inputs.CouplerState <-> Inputs/CouplerState
//     PlcTask Inputs/GVL_iXlinker.EtherCAT_Master_BKCUCX.Beckhoff_BKxxxx.Beckhoff_BKxxxxEK1122.A_0004_BK1120_0000_0017.Outputs.CouplerCtrl <-> Outputs/CouplerCtrl
//     PlcTask Inputs/GVL_iXlinker.EtherCAT_Master_BKCUCX.Beckhoff_BKxxxx.Beckhoff_BKxxxxEK1122.A_0004_BK1120_0000_0017.WcState.WcState <-> WcState/WcState
//     PlcTask Inputs/GVL_iXlinker.EtherCAT_Master_BKCUCX.Beckhoff_BKxxxx.Beckhoff_BKxxxxEK1122.A_0004_BK1120_0000_0017.WcState.InputToggle <-> WcState/InputToggle
//     PlcTask Inputs/GVL_iXlinker.EtherCAT_Master_BKCUCX.Beckhoff_BKxxxx.Beckhoff_BKxxxxEK1122.A_0004_BK1120_0000_0017.InfoData.AdsAddr <-> InfoData/AdsAddr
//     PlcTask Inputs/GVL_iXlinker.EtherCAT_Master_BKCUCX.Beckhoff_BKxxxx.Beckhoff_BKxxxxEK1122.A_0004_BK1120_0000_0017.InfoData.AoeNetId <-> InfoData/AoeNetId
//     PlcTask Inputs/GVL_iXlinker.EtherCAT_Master_BKCUCX.Beckhoff_BKxxxx.Beckhoff_BKxxxxEK1122.A_0004_BK1120_0000_0017.InfoData.State <-> InfoData/State
//   PLC/PLC Instance <-> EtherCAT Master BKCUCX/Beckhoff BKxxxx/Beckhoff BKxxxxEK1122/A_0004(BK1120-0000-0017)/Term 377 (KL1002)
//     PlcTask Inputs/GVL_iXlinker.EtherCAT_Master_BKCUCX.Beckhoff_BKxxxx.Beckhoff_BKxxxxEK1122.A_0004_BK1120_0000_0017.Term_377_KL1002.Channel_1.Input <-> Channel 1/Input
//     PlcTask Inputs/GVL_iXlinker.EtherCAT_Master_BKCUCX.Beckhoff_BKxxxx.Beckhoff_BKxxxxEK1122.A_0004_BK1120_0000_0017.Term_377_KL1002.Channel_2.Input <-> Channel 2/Input
//   PLC/PLC Instance <-> EtherCAT Master BKCUCX/Beckhoff BKxxxx/Beckhoff BKxxxxEK1122/A_0005(BK1120-0000-0018)
//     PlcTask Inputs/GVL_iXlinker.EtherCAT_Master_BKCUCX.Beckhoff_BKxxxx.Beckhoff_BKxxxxEK1122.A_0005_BK1120_0000_0018.Inputs.CouplerState <-> Inputs/CouplerState
//     PlcTask Inputs/GVL_iXlinker.EtherCAT_Master_BKCUCX.Beckhoff_BKxxxx.Beckhoff_BKxxxxEK1122.A_0005_BK1120_0000_0018.Outputs.CouplerCtrl <-> Outputs/CouplerCtrl
//     PlcTask Inputs/GVL_iXlinker.EtherCAT_Master_BKCUCX.Beckhoff_BKxxxx.Beckhoff_BKxxxxEK1122.A_0005_BK1120_0000_0018.WcState.WcState <-> WcState/WcState
//     PlcTask Inputs/GVL_iXlinker.EtherCAT_Master_BKCUCX.Beckhoff_BKxxxx.Beckhoff_BKxxxxEK1122.A_0005_BK1120_0000_0018.WcState.InputToggle <-> WcState/InputToggle
//     PlcTask Inputs/GVL_iXlinker.EtherCAT_Master_BKCUCX.Beckhoff_BKxxxx.Beckhoff_BKxxxxEK1122.A_0005_BK1120_0000_0018.InfoData.AdsAddr <-> InfoData/AdsAddr
//     PlcTask Inputs/GVL_iXlinker.EtherCAT_Master_BKCUCX.Beckhoff_BKxxxx.Beckhoff_BKxxxxEK1122.A_0005_BK1120_0000_0018.InfoData.AoeNetId <-> InfoData/AoeNetId
//     PlcTask Inputs/GVL_iXlinker.EtherCAT_Master_BKCUCX.Beckhoff_BKxxxx.Beckhoff_BKxxxxEK1122.A_0005_BK1120_0000_0018.InfoData.State <-> InfoData/State
//   PLC/PLC Instance <-> EtherCAT Master BKCUCX/Beckhoff BKxxxx/Beckhoff BKxxxxEK1122/A_0005(BK1120-0000-0018)/Term 378 (KL1002)
//     PlcTask Inputs/GVL_iXlinker.EtherCAT_Master_BKCUCX.Beckhoff_BKxxxx.Beckhoff_BKxxxxEK1122.A_0005_BK1120_0000_0018.Term_378_KL1002.Channel_1.Input <-> Channel 1/Input
//     PlcTask Inputs/GVL_iXlinker.EtherCAT_Master_BKCUCX.Beckhoff_BKxxxx.Beckhoff_BKxxxxEK1122.A_0005_BK1120_0000_0018.Term_378_KL1002.Channel_2.Input <-> Channel 2/Input
//   PLC/PLC Instance <-> EtherCAT Master BKCUCX/Beckhoff BKxxxx/Beckhoff BKxxxxEK1122/A_0006(BK1120-0000-0019)
//     PlcTask Inputs/GVL_iXlinker.EtherCAT_Master_BKCUCX.Beckhoff_BKxxxx.Beckhoff_BKxxxxEK1122.A_0006_BK1120_0000_0019.Inputs.CouplerState <-> Inputs/CouplerState
//     PlcTask Inputs/GVL_iXlinker.EtherCAT_Master_BKCUCX.Beckhoff_BKxxxx.Beckhoff_BKxxxxEK1122.A_0006_BK1120_0000_0019.Outputs.CouplerCtrl <-> Outputs/CouplerCtrl
//     PlcTask Inputs/GVL_iXlinker.EtherCAT_Master_BKCUCX.Beckhoff_BKxxxx.Beckhoff_BKxxxxEK1122.A_0006_BK1120_0000_0019.WcState.WcState <-> WcState/WcState
//     PlcTask Inputs/GVL_iXlinker.EtherCAT_Master_BKCUCX.Beckhoff_BKxxxx.Beckhoff_BKxxxxEK1122.A_0006_BK1120_0000_0019.WcState.InputToggle <-> WcState/InputToggle
//     PlcTask Inputs/GVL_iXlinker.EtherCAT_Master_BKCUCX.Beckhoff_BKxxxx.Beckhoff_BKxxxxEK1122.A_0006_BK1120_0000_0019.InfoData.AdsAddr <-> InfoData/AdsAddr
//     PlcTask Inputs/GVL_iXlinker.EtherCAT_Master_BKCUCX.Beckhoff_BKxxxx.Beckhoff_BKxxxxEK1122.A_0006_BK1120_0000_0019.InfoData.AoeNetId <-> InfoData/AoeNetId
//     PlcTask Inputs/GVL_iXlinker.EtherCAT_Master_BKCUCX.Beckhoff_BKxxxx.Beckhoff_BKxxxxEK1122.A_0006_BK1120_0000_0019.InfoData.State <-> InfoData/State
//   PLC/PLC Instance <-> EtherCAT Master BKCUCX/Beckhoff BKxxxx/Beckhoff BKxxxxEK1122/A_0006(BK1120-0000-0019)/Term 379 (KL1002)
//     PlcTask Inputs/GVL_iXlinker.EtherCAT_Master_BKCUCX.Beckhoff_BKxxxx.Beckhoff_BKxxxxEK1122.A_0006_BK1120_0000_0019.Term_379_KL1002.Channel_1.Input <-> Channel 1/Input
//     PlcTask Inputs/GVL_iXlinker.EtherCAT_Master_BKCUCX.Beckhoff_BKxxxx.Beckhoff_BKxxxxEK1122.A_0006_BK1120_0000_0019.Term_379_KL1002.Channel_2.Input <-> Channel 2/Input
//   PLC/PLC Instance <-> EtherCAT Master BKCUCX/Beckhoff BKxxxx/Beckhoff BKxxxxEK1122/A_0007(BK1120-0000-0020)
//     PlcTask Inputs/GVL_iXlinker.EtherCAT_Master_BKCUCX.Beckhoff_BKxxxx.Beckhoff_BKxxxxEK1122.A_0007_BK1120_0000_0020.Inputs.CouplerState <-> Inputs/CouplerState
//     PlcTask Inputs/GVL_iXlinker.EtherCAT_Master_BKCUCX.Beckhoff_BKxxxx.Beckhoff_BKxxxxEK1122.A_0007_BK1120_0000_0020.Outputs.CouplerCtrl <-> Outputs/CouplerCtrl
//     PlcTask Inputs/GVL_iXlinker.EtherCAT_Master_BKCUCX.Beckhoff_BKxxxx.Beckhoff_BKxxxxEK1122.A_0007_BK1120_0000_0020.WcState.WcState <-> WcState/WcState
//     PlcTask Inputs/GVL_iXlinker.EtherCAT_Master_BKCUCX.Beckhoff_BKxxxx.Beckhoff_BKxxxxEK1122.A_0007_BK1120_0000_0020.WcState.InputToggle <-> WcState/InputToggle
//     PlcTask Inputs/GVL_iXlinker.EtherCAT_Master_BKCUCX.Beckhoff_BKxxxx.Beckhoff_BKxxxxEK1122.A_0007_BK1120_0000_0020.InfoData.AdsAddr <-> InfoData/AdsAddr
//     PlcTask Inputs/GVL_iXlinker.EtherCAT_Master_BKCUCX.Beckhoff_BKxxxx.Beckhoff_BKxxxxEK1122.A_0007_BK1120_0000_0020.InfoData.AoeNetId <-> InfoData/AoeNetId
//     PlcTask Inputs/GVL_iXlinker.EtherCAT_Master_BKCUCX.Beckhoff_BKxxxx.Beckhoff_BKxxxxEK1122.A_0007_BK1120_0000_0020.InfoData.State <-> InfoData/State
//   PLC/PLC Instance <-> EtherCAT Master BKCUCX/Beckhoff BKxxxx/Beckhoff BKxxxxEK1122/A_0007(BK1120-0000-0020)/Term 380 (KL1002)
//     PlcTask Inputs/GVL_iXlinker.EtherCAT_Master_BKCUCX.Beckhoff_BKxxxx.Beckhoff_BKxxxxEK1122.A_0007_BK1120_0000_0020.Term_380_KL1002.Channel_1.Input <-> Channel 1/Input
//     PlcTask Inputs/GVL_iXlinker.EtherCAT_Master_BKCUCX.Beckhoff_BKxxxx.Beckhoff_BKxxxxEK1122.A_0007_BK1120_0000_0020.Term_380_KL1002.Channel_2.Input <-> Channel 2/Input
//   PLC/PLC Instance <-> EtherCAT Master BKCUCX/Beckhoff BKxxxx/Beckhoff BKxxxxEK1122/A_0008(BK1120-0000-0021)
//     PlcTask Inputs/GVL_iXlinker.EtherCAT_Master_BKCUCX.Beckhoff_BKxxxx.Beckhoff_BKxxxxEK1122.A_0008_BK1120_0000_0021.Inputs.CouplerState <-> Inputs/CouplerState
//     PlcTask Inputs/GVL_iXlinker.EtherCAT_Master_BKCUCX.Beckhoff_BKxxxx.Beckhoff_BKxxxxEK1122.A_0008_BK1120_0000_0021.Outputs.CouplerCtrl <-> Outputs/CouplerCtrl
//     PlcTask Inputs/GVL_iXlinker.EtherCAT_Master_BKCUCX.Beckhoff_BKxxxx.Beckhoff_BKxxxxEK1122.A_0008_BK1120_0000_0021.WcState.WcState <-> WcState/WcState
//     PlcTask Inputs/GVL_iXlinker.EtherCAT_Master_BKCUCX.Beckhoff_BKxxxx.Beckhoff_BKxxxxEK1122.A_0008_BK1120_0000_0021.WcState.InputToggle <-> WcState/InputToggle
//     PlcTask Inputs/GVL_iXlinker.EtherCAT_Master_BKCUCX.Beckhoff_BKxxxx.Beckhoff_BKxxxxEK1122.A_0008_BK1120_0000_0021.InfoData.AdsAddr <-> InfoData/AdsAddr
//     PlcTask Inputs/GVL_iXlinker.EtherCAT_Master_BKCUCX.Beckhoff_BKxxxx.Beckhoff_BKxxxxEK1122.A_0008_BK1120_0000_0021.InfoData.AoeNetId <-> InfoData/AoeNetId
//     PlcTask Inputs/GVL_iXlinker.EtherCAT_Master_BKCUCX.Beckhoff_BKxxxx.Beckhoff_BKxxxxEK1122.A_0008_BK1120_0000_0021.InfoData.State <-> InfoData/State
//   PLC/PLC Instance <-> EtherCAT Master BKCUCX/Beckhoff BKxxxx/Beckhoff BKxxxxEK1122/A_0008(BK1120-0000-0021)/Term 381 (KL1002)
//     PlcTask Inputs/GVL_iXlinker.EtherCAT_Master_BKCUCX.Beckhoff_BKxxxx.Beckhoff_BKxxxxEK1122.A_0008_BK1120_0000_0021.Term_381_KL1002.Channel_1.Input <-> Channel 1/Input
//     PlcTask Inputs/GVL_iXlinker.EtherCAT_Master_BKCUCX.Beckhoff_BKxxxx.Beckhoff_BKxxxxEK1122.A_0008_BK1120_0000_0021.Term_381_KL1002.Channel_2.Input <-> Channel 2/Input
//   PLC/PLC Instance <-> EtherCAT Master BKCUCX/Beckhoff BKxxxx/Beckhoff BKxxxxEK1122/A_0009(CPXXXX-BK1150-0016)
//     PlcTask Inputs/GVL_iXlinker.EtherCAT_Master_BKCUCX.Beckhoff_BKxxxx.Beckhoff_BKxxxxEK1122.A_0009_CPXXXX_BK1150_0016.Inputs.CouplerState <-> Inputs/CouplerState
//     PlcTask Inputs/GVL_iXlinker.EtherCAT_Master_BKCUCX.Beckhoff_BKxxxx.Beckhoff_BKxxxxEK1122.A_0009_CPXXXX_BK1150_0016.Outputs.CouplerCtrl <-> Outputs/CouplerCtrl
//     PlcTask Inputs/GVL_iXlinker.EtherCAT_Master_BKCUCX.Beckhoff_BKxxxx.Beckhoff_BKxxxxEK1122.A_0009_CPXXXX_BK1150_0016.WcState.WcState <-> WcState/WcState
//     PlcTask Inputs/GVL_iXlinker.EtherCAT_Master_BKCUCX.Beckhoff_BKxxxx.Beckhoff_BKxxxxEK1122.A_0009_CPXXXX_BK1150_0016.WcState.InputToggle <-> WcState/InputToggle
//     PlcTask Inputs/GVL_iXlinker.EtherCAT_Master_BKCUCX.Beckhoff_BKxxxx.Beckhoff_BKxxxxEK1122.A_0009_CPXXXX_BK1150_0016.InfoData.AdsAddr <-> InfoData/AdsAddr
//     PlcTask Inputs/GVL_iXlinker.EtherCAT_Master_BKCUCX.Beckhoff_BKxxxx.Beckhoff_BKxxxxEK1122.A_0009_CPXXXX_BK1150_0016.InfoData.AoeNetId <-> InfoData/AoeNetId
//     PlcTask Inputs/GVL_iXlinker.EtherCAT_Master_BKCUCX.Beckhoff_BKxxxx.Beckhoff_BKxxxxEK1122.A_0009_CPXXXX_BK1150_0016.InfoData.State <-> InfoData/State
//   PLC/PLC Instance <-> EtherCAT Master BKCUCX/Beckhoff BKxxxx/Beckhoff BKxxxxEK1122/A_0009(CPXXXX-BK1150-0016)/Term 382 (KL1002)
//     PlcTask Inputs/GVL_iXlinker.EtherCAT_Master_BKCUCX.Beckhoff_BKxxxx.Beckhoff_BKxxxxEK1122.A_0009_CPXXXX_BK1150_0016.Term_382_KL1002.Channel_1.Input <-> Channel 1/Input
//     PlcTask Inputs/GVL_iXlinker.EtherCAT_Master_BKCUCX.Beckhoff_BKxxxx.Beckhoff_BKxxxxEK1122.A_0009_CPXXXX_BK1150_0016.Term_382_KL1002.Channel_2.Input <-> Channel 2/Input
//   PLC/PLC Instance <-> EtherCAT Master BKCUCX/Beckhoff BKxxxx/Beckhoff BKxxxxEK1122/A_0010(BK1150-0000-0016)
//     PlcTask Inputs/GVL_iXlinker.EtherCAT_Master_BKCUCX.Beckhoff_BKxxxx.Beckhoff_BKxxxxEK1122.A_0010_BK1150_0000_0016.Inputs.CouplerState <-> Inputs/CouplerState
//     PlcTask Inputs/GVL_iXlinker.EtherCAT_Master_BKCUCX.Beckhoff_BKxxxx.Beckhoff_BKxxxxEK1122.A_0010_BK1150_0000_0016.Outputs.CouplerCtrl <-> Outputs/CouplerCtrl
//     PlcTask Inputs/GVL_iXlinker.EtherCAT_Master_BKCUCX.Beckhoff_BKxxxx.Beckhoff_BKxxxxEK1122.A_0010_BK1150_0000_0016.WcState.WcState <-> WcState/WcState
//     PlcTask Inputs/GVL_iXlinker.EtherCAT_Master_BKCUCX.Beckhoff_BKxxxx.Beckhoff_BKxxxxEK1122.A_0010_BK1150_0000_0016.WcState.InputToggle <-> WcState/InputToggle
//     PlcTask Inputs/GVL_iXlinker.EtherCAT_Master_BKCUCX.Beckhoff_BKxxxx.Beckhoff_BKxxxxEK1122.A_0010_BK1150_0000_0016.InfoData.AdsAddr <-> InfoData/AdsAddr
//     PlcTask Inputs/GVL_iXlinker.EtherCAT_Master_BKCUCX.Beckhoff_BKxxxx.Beckhoff_BKxxxxEK1122.A_0010_BK1150_0000_0016.InfoData.AoeNetId <-> InfoData/AoeNetId
//     PlcTask Inputs/GVL_iXlinker.EtherCAT_Master_BKCUCX.Beckhoff_BKxxxx.Beckhoff_BKxxxxEK1122.A_0010_BK1150_0000_0016.InfoData.State <-> InfoData/State
//   PLC/PLC Instance <-> EtherCAT Master BKCUCX/Beckhoff BKxxxx/Beckhoff BKxxxxEK1122/A_0010(BK1150-0000-0016)/Term 383 (KL1002)
//     PlcTask Inputs/GVL_iXlinker.EtherCAT_Master_BKCUCX.Beckhoff_BKxxxx.Beckhoff_BKxxxxEK1122.A_0010_BK1150_0000_0016.Term_383_KL1002.Channel_1.Input <-> Channel 1/Input
//     PlcTask Inputs/GVL_iXlinker.EtherCAT_Master_BKCUCX.Beckhoff_BKxxxx.Beckhoff_BKxxxxEK1122.A_0010_BK1150_0000_0016.Term_383_KL1002.Channel_2.Input <-> Channel 2/Input
//   PLC/PLC Instance <-> EtherCAT Master BKCUCX/Beckhoff BKxxxx/Beckhoff BKxxxxEK1122/A_0011(BK1150-0000-0017)
//     PlcTask Inputs/GVL_iXlinker.EtherCAT_Master_BKCUCX.Beckhoff_BKxxxx.Beckhoff_BKxxxxEK1122.A_0011_BK1150_0000_0017.Inputs.CouplerState <-> Inputs/CouplerState
//     PlcTask Inputs/GVL_iXlinker.EtherCAT_Master_BKCUCX.Beckhoff_BKxxxx.Beckhoff_BKxxxxEK1122.A_0011_BK1150_0000_0017.Outputs.CouplerCtrl <-> Outputs/CouplerCtrl
//     PlcTask Inputs/GVL_iXlinker.EtherCAT_Master_BKCUCX.Beckhoff_BKxxxx.Beckhoff_BKxxxxEK1122.A_0011_BK1150_0000_0017.WcState.WcState <-> WcState/WcState
//     PlcTask Inputs/GVL_iXlinker.EtherCAT_Master_BKCUCX.Beckhoff_BKxxxx.Beckhoff_BKxxxxEK1122.A_0011_BK1150_0000_0017.WcState.InputToggle <-> WcState/InputToggle
//     PlcTask Inputs/GVL_iXlinker.EtherCAT_Master_BKCUCX.Beckhoff_BKxxxx.Beckhoff_BKxxxxEK1122.A_0011_BK1150_0000_0017.InfoData.AdsAddr <-> InfoData/AdsAddr
//     PlcTask Inputs/GVL_iXlinker.EtherCAT_Master_BKCUCX.Beckhoff_BKxxxx.Beckhoff_BKxxxxEK1122.A_0011_BK1150_0000_0017.InfoData.AoeNetId <-> InfoData/AoeNetId
//     PlcTask Inputs/GVL_iXlinker.EtherCAT_Master_BKCUCX.Beckhoff_BKxxxx.Beckhoff_BKxxxxEK1122.A_0011_BK1150_0000_0017.InfoData.State <-> InfoData/State
//   PLC/PLC Instance <-> EtherCAT Master BKCUCX/Beckhoff BKxxxx/Beckhoff BKxxxxEK1122/A_0011(BK1150-0000-0017)/Term 384 (KL1002)
//     PlcTask Inputs/GVL_iXlinker.EtherCAT_Master_BKCUCX.Beckhoff_BKxxxx.Beckhoff_BKxxxxEK1122.A_0011_BK1150_0000_0017.Term_384_KL1002.Channel_1.Input <-> Channel 1/Input
//     PlcTask Inputs/GVL_iXlinker.EtherCAT_Master_BKCUCX.Beckhoff_BKxxxx.Beckhoff_BKxxxxEK1122.A_0011_BK1150_0000_0017.Term_384_KL1002.Channel_2.Input <-> Channel 2/Input
//   PLC/PLC Instance <-> EtherCAT Master BKCUCX/Beckhoff BKxxxx/Beckhoff BKxxxxEK1122/A_0012(BK1150-0000-0018)
//     PlcTask Inputs/GVL_iXlinker.EtherCAT_Master_BKCUCX.Beckhoff_BKxxxx.Beckhoff_BKxxxxEK1122.A_0012_BK1150_0000_0018.Inputs.CouplerState <-> Inputs/CouplerState
//     PlcTask Inputs/GVL_iXlinker.EtherCAT_Master_BKCUCX.Beckhoff_BKxxxx.Beckhoff_BKxxxxEK1122.A_0012_BK1150_0000_0018.Outputs.CouplerCtrl <-> Outputs/CouplerCtrl
//     PlcTask Inputs/GVL_iXlinker.EtherCAT_Master_BKCUCX.Beckhoff_BKxxxx.Beckhoff_BKxxxxEK1122.A_0012_BK1150_0000_0018.WcState.WcState <-> WcState/WcState
//     PlcTask Inputs/GVL_iXlinker.EtherCAT_Master_BKCUCX.Beckhoff_BKxxxx.Beckhoff_BKxxxxEK1122.A_0012_BK1150_0000_0018.WcState.InputToggle <-> WcState/InputToggle
//     PlcTask Inputs/GVL_iXlinker.EtherCAT_Master_BKCUCX.Beckhoff_BKxxxx.Beckhoff_BKxxxxEK1122.A_0012_BK1150_0000_0018.InfoData.AdsAddr <-> InfoData/AdsAddr
//     PlcTask Inputs/GVL_iXlinker.EtherCAT_Master_BKCUCX.Beckhoff_BKxxxx.Beckhoff_BKxxxxEK1122.A_0012_BK1150_0000_0018.InfoData.AoeNetId <-> InfoData/AoeNetId
//     PlcTask Inputs/GVL_iXlinker.EtherCAT_Master_BKCUCX.Beckhoff_BKxxxx.Beckhoff_BKxxxxEK1122.A_0012_BK1150_0000_0018.InfoData.State <-> InfoData/State
//   PLC/PLC Instance <-> EtherCAT Master BKCUCX/Beckhoff BKxxxx/Beckhoff BKxxxxEK1122/A_0012(BK1150-0000-0018)/Term 385 (KL1002)
//     PlcTask Inputs/GVL_iXlinker.EtherCAT_Master_BKCUCX.Beckhoff_BKxxxx.Beckhoff_BKxxxxEK1122.A_0012_BK1150_0000_0018.Term_385_KL1002.Channel_1.Input <-> Channel 1/Input
//     PlcTask Inputs/GVL_iXlinker.EtherCAT_Master_BKCUCX.Beckhoff_BKxxxx.Beckhoff_BKxxxxEK1122.A_0012_BK1150_0000_0018.Term_385_KL1002.Channel_2.Input <-> Channel 2/Input
//   PLC/PLC Instance <-> EtherCAT Master BKCUCX/Beckhoff BKxxxx/Beckhoff BKxxxxEK1122/A_0013(BK1150-0000-0019)
//     PlcTask Inputs/GVL_iXlinker.EtherCAT_Master_BKCUCX.Beckhoff_BKxxxx.Beckhoff_BKxxxxEK1122.A_0013_BK1150_0000_0019.Inputs.CouplerState <-> Inputs/CouplerState
//     PlcTask Inputs/GVL_iXlinker.EtherCAT_Master_BKCUCX.Beckhoff_BKxxxx.Beckhoff_BKxxxxEK1122.A_0013_BK1150_0000_0019.Outputs.CouplerCtrl <-> Outputs/CouplerCtrl
//     PlcTask Inputs/GVL_iXlinker.EtherCAT_Master_BKCUCX.Beckhoff_BKxxxx.Beckhoff_BKxxxxEK1122.A_0013_BK1150_0000_0019.WcState.WcState <-> WcState/WcState
//     PlcTask Inputs/GVL_iXlinker.EtherCAT_Master_BKCUCX.Beckhoff_BKxxxx.Beckhoff_BKxxxxEK1122.A_0013_BK1150_0000_0019.WcState.InputToggle <-> WcState/InputToggle
//     PlcTask Inputs/GVL_iXlinker.EtherCAT_Master_BKCUCX.Beckhoff_BKxxxx.Beckhoff_BKxxxxEK1122.A_0013_BK1150_0000_0019.InfoData.AdsAddr <-> InfoData/AdsAddr
//     PlcTask Inputs/GVL_iXlinker.EtherCAT_Master_BKCUCX.Beckhoff_BKxxxx.Beckhoff_BKxxxxEK1122.A_0013_BK1150_0000_0019.InfoData.AoeNetId <-> InfoData/AoeNetId
//     PlcTask Inputs/GVL_iXlinker.EtherCAT_Master_BKCUCX.Beckhoff_BKxxxx.Beckhoff_BKxxxxEK1122.A_0013_BK1150_0000_0019.InfoData.State <-> InfoData/State
//   PLC/PLC Instance <-> EtherCAT Master BKCUCX/Beckhoff BKxxxx/Beckhoff BKxxxxEK1122/A_0013(BK1150-0000-0019)/Term 386 (KL1002)
//     PlcTask Inputs/GVL_iXlinker.EtherCAT_Master_BKCUCX.Beckhoff_BKxxxx.Beckhoff_BKxxxxEK1122.A_0013_BK1150_0000_0019.Term_386_KL1002.Channel_1.Input <-> Channel 1/Input
//     PlcTask Inputs/GVL_iXlinker.EtherCAT_Master_BKCUCX.Beckhoff_BKxxxx.Beckhoff_BKxxxxEK1122.A_0013_BK1150_0000_0019.Term_386_KL1002.Channel_2.Input <-> Channel 2/Input
//   PLC/PLC Instance <-> EtherCAT Master BKCUCX/Beckhoff BKxxxx/Beckhoff BKxxxxEK1122/Term 19 (EK1100)
//     PlcTask Inputs/GVL_iXlinker.EtherCAT_Master_BKCUCX.Beckhoff_BKxxxx.Beckhoff_BKxxxxEK1122.Term_19_EK1100.InfoData.State <-> InfoData/State
//   PLC/PLC Instance <-> EtherCAT Master BKCUCX/Beckhoff BKxxxx/Beckhoff BKxxxxEK1122/Term 19 (EK1100)/A_0016(BK1250-0000-0017)
//     PlcTask Inputs/GVL_iXlinker.EtherCAT_Master_BKCUCX.Beckhoff_BKxxxx.Beckhoff_BKxxxxEK1122.Term_19_EK1100.A_0016_BK1250_0000_0017.Inputs.CouplerState <-> Inputs/CouplerState
//     PlcTask Inputs/GVL_iXlinker.EtherCAT_Master_BKCUCX.Beckhoff_BKxxxx.Beckhoff_BKxxxxEK1122.Term_19_EK1100.A_0016_BK1250_0000_0017.Outputs.CouplerCtrl <-> Outputs/CouplerCtrl
//     PlcTask Inputs/GVL_iXlinker.EtherCAT_Master_BKCUCX.Beckhoff_BKxxxx.Beckhoff_BKxxxxEK1122.Term_19_EK1100.A_0016_BK1250_0000_0017.WcState.WcState <-> WcState/WcState
//     PlcTask Inputs/GVL_iXlinker.EtherCAT_Master_BKCUCX.Beckhoff_BKxxxx.Beckhoff_BKxxxxEK1122.Term_19_EK1100.A_0016_BK1250_0000_0017.WcState.InputToggle <-> WcState/InputToggle
//     PlcTask Inputs/GVL_iXlinker.EtherCAT_Master_BKCUCX.Beckhoff_BKxxxx.Beckhoff_BKxxxxEK1122.Term_19_EK1100.A_0016_BK1250_0000_0017.InfoData.AdsAddr <-> InfoData/AdsAddr
//     PlcTask Inputs/GVL_iXlinker.EtherCAT_Master_BKCUCX.Beckhoff_BKxxxx.Beckhoff_BKxxxxEK1122.Term_19_EK1100.A_0016_BK1250_0000_0017.InfoData.AoeNetId <-> InfoData/AoeNetId
//     PlcTask Inputs/GVL_iXlinker.EtherCAT_Master_BKCUCX.Beckhoff_BKxxxx.Beckhoff_BKxxxxEK1122.Term_19_EK1100.A_0016_BK1250_0000_0017.InfoData.State <-> InfoData/State
//   PLC/PLC Instance <-> EtherCAT Master BKCUCX/Beckhoff BKxxxx/Beckhoff BKxxxxEK1122/Term 19 (EK1100)/A_0016(BK1250-0000-0017)/Term 387 (KL1002)
//     PlcTask Inputs/GVL_iXlinker.EtherCAT_Master_BKCUCX.Beckhoff_BKxxxx.Beckhoff_BKxxxxEK1122.Term_19_EK1100.A_0016_BK1250_0000_0017.Term_387_KL1002.Channel_1.Input <-> Channel 1/Input
//     PlcTask Inputs/GVL_iXlinker.EtherCAT_Master_BKCUCX.Beckhoff_BKxxxx.Beckhoff_BKxxxxEK1122.Term_19_EK1100.A_0016_BK1250_0000_0017.Term_387_KL1002.Channel_2.Input <-> Channel 2/Input
//   PLC/PLC Instance <-> EtherCAT Master BKCUCX/Beckhoff BKxxxx/Beckhoff BKxxxxEK1122/Term 23 (EK1100)
//     PlcTask Inputs/GVL_iXlinker.EtherCAT_Master_BKCUCX.Beckhoff_BKxxxx.Beckhoff_BKxxxxEK1122.Term_23_EK1100.InfoData.State <-> InfoData/State
//   PLC/PLC Instance <-> EtherCAT Master BKCUCX/Beckhoff BKxxxx/Beckhoff BKxxxxEK1122/Term 23 (EK1100)/A_0018(BK1250-0000-0019)
//     PlcTask Inputs/GVL_iXlinker.EtherCAT_Master_BKCUCX.Beckhoff_BKxxxx.Beckhoff_BKxxxxEK1122.Term_23_EK1100.A_0018_BK1250_0000_0019.Inputs.CouplerState <-> Inputs/CouplerState
//     PlcTask Inputs/GVL_iXlinker.EtherCAT_Master_BKCUCX.Beckhoff_BKxxxx.Beckhoff_BKxxxxEK1122.Term_23_EK1100.A_0018_BK1250_0000_0019.Outputs.CouplerCtrl <-> Outputs/CouplerCtrl
//     PlcTask Inputs/GVL_iXlinker.EtherCAT_Master_BKCUCX.Beckhoff_BKxxxx.Beckhoff_BKxxxxEK1122.Term_23_EK1100.A_0018_BK1250_0000_0019.WcState.WcState <-> WcState/WcState
//     PlcTask Inputs/GVL_iXlinker.EtherCAT_Master_BKCUCX.Beckhoff_BKxxxx.Beckhoff_BKxxxxEK1122.Term_23_EK1100.A_0018_BK1250_0000_0019.WcState.InputToggle <-> WcState/InputToggle
//     PlcTask Inputs/GVL_iXlinker.EtherCAT_Master_BKCUCX.Beckhoff_BKxxxx.Beckhoff_BKxxxxEK1122.Term_23_EK1100.A_0018_BK1250_0000_0019.InfoData.AdsAddr <-> InfoData/AdsAddr
//     PlcTask Inputs/GVL_iXlinker.EtherCAT_Master_BKCUCX.Beckhoff_BKxxxx.Beckhoff_BKxxxxEK1122.Term_23_EK1100.A_0018_BK1250_0000_0019.InfoData.AoeNetId <-> InfoData/AoeNetId
//     PlcTask Inputs/GVL_iXlinker.EtherCAT_Master_BKCUCX.Beckhoff_BKxxxx.Beckhoff_BKxxxxEK1122.Term_23_EK1100.A_0018_BK1250_0000_0019.InfoData.State <-> InfoData/State
//   PLC/PLC Instance <-> EtherCAT Master BKCUCX/Beckhoff BKxxxx/Beckhoff BKxxxxEK1122/Term 23 (EK1100)/A_0018(BK1250-0000-0019)/Term 388 (KL1002)
//     PlcTask Inputs/GVL_iXlinker.EtherCAT_Master_BKCUCX.Beckhoff_BKxxxx.Beckhoff_BKxxxxEK1122.Term_23_EK1100.A_0018_BK1250_0000_0019.Term_388_KL1002.Channel_1.Input <-> Channel 1/Input
//     PlcTask Inputs/GVL_iXlinker.EtherCAT_Master_BKCUCX.Beckhoff_BKxxxx.Beckhoff_BKxxxxEK1122.Term_23_EK1100.A_0018_BK1250_0000_0019.Term_388_KL1002.Channel_2.Input <-> Channel 2/Input
//   PLC/PLC Instance <-> EtherCAT Master BKCUCX/Beckhoff BKxxxx/Beckhoff BKxxxxEK1122/Term 21 (EK1100)
//     PlcTask Inputs/GVL_iXlinker.EtherCAT_Master_BKCUCX.Beckhoff_BKxxxx.Beckhoff_BKxxxxEK1122.Term_21_EK1100.InfoData.State <-> InfoData/State
//   PLC/PLC Instance <-> EtherCAT Master BKCUCX/Beckhoff BKxxxx/Beckhoff BKxxxxEK1122/Term 21 (EK1100)/A_0017(BK1250-0000-0018)
//     PlcTask Inputs/GVL_iXlinker.EtherCAT_Master_BKCUCX.Beckhoff_BKxxxx.Beckhoff_BKxxxxEK1122.Term_21_EK1100.A_0017_BK1250_0000_0018.Inputs.CouplerState <-> Inputs/CouplerState
//     PlcTask Inputs/GVL_iXlinker.EtherCAT_Master_BKCUCX.Beckhoff_BKxxxx.Beckhoff_BKxxxxEK1122.Term_21_EK1100.A_0017_BK1250_0000_0018.Outputs.CouplerCtrl <-> Outputs/CouplerCtrl
//     PlcTask Inputs/GVL_iXlinker.EtherCAT_Master_BKCUCX.Beckhoff_BKxxxx.Beckhoff_BKxxxxEK1122.Term_21_EK1100.A_0017_BK1250_0000_0018.WcState.WcState <-> WcState/WcState
//     PlcTask Inputs/GVL_iXlinker.EtherCAT_Master_BKCUCX.Beckhoff_BKxxxx.Beckhoff_BKxxxxEK1122.Term_21_EK1100.A_0017_BK1250_0000_0018.WcState.InputToggle <-> WcState/InputToggle
//     PlcTask Inputs/GVL_iXlinker.EtherCAT_Master_BKCUCX.Beckhoff_BKxxxx.Beckhoff_BKxxxxEK1122.Term_21_EK1100.A_0017_BK1250_0000_0018.InfoData.AdsAddr <-> InfoData/AdsAddr
//     PlcTask Inputs/GVL_iXlinker.EtherCAT_Master_BKCUCX.Beckhoff_BKxxxx.Beckhoff_BKxxxxEK1122.Term_21_EK1100.A_0017_BK1250_0000_0018.InfoData.AoeNetId <-> InfoData/AoeNetId
//     PlcTask Inputs/GVL_iXlinker.EtherCAT_Master_BKCUCX.Beckhoff_BKxxxx.Beckhoff_BKxxxxEK1122.Term_21_EK1100.A_0017_BK1250_0000_0018.InfoData.State <-> InfoData/State
//   PLC/PLC Instance <-> EtherCAT Master BKCUCX/Beckhoff BKxxxx/Beckhoff BKxxxxEK1122/Term 21 (EK1100)/A_0017(BK1250-0000-0018)/Term 389 (KL1002)
//     PlcTask Inputs/GVL_iXlinker.EtherCAT_Master_BKCUCX.Beckhoff_BKxxxx.Beckhoff_BKxxxxEK1122.Term_21_EK1100.A_0017_BK1250_0000_0018.Term_389_KL1002.Channel_1.Input <-> Channel 1/Input
//     PlcTask Inputs/GVL_iXlinker.EtherCAT_Master_BKCUCX.Beckhoff_BKxxxx.Beckhoff_BKxxxxEK1122.Term_21_EK1100.A_0017_BK1250_0000_0018.Term_389_KL1002.Channel_2.Input <-> Channel 2/Input
//   PLC/PLC Instance <-> EtherCAT Master BKCUCX/Beckhoff BKxxxx/Beckhoff BKxxxxEK1122/A_0019(IL2300-B110-0016)
//     PlcTask Inputs/GVL_iXlinker.EtherCAT_Master_BKCUCX.Beckhoff_BKxxxx.Beckhoff_BKxxxxEK1122.A_0019_IL2300_B110_0016.Inputs.CouplerState <-> Inputs/CouplerState
//     PlcTask Inputs/GVL_iXlinker.EtherCAT_Master_BKCUCX.Beckhoff_BKxxxx.Beckhoff_BKxxxxEK1122.A_0019_IL2300_B110_0016.Outputs.CouplerCtrl <-> Outputs/CouplerCtrl
//     PlcTask Inputs/GVL_iXlinker.EtherCAT_Master_BKCUCX.Beckhoff_BKxxxx.Beckhoff_BKxxxxEK1122.A_0019_IL2300_B110_0016.WcState.WcState <-> WcState/WcState
//     PlcTask Inputs/GVL_iXlinker.EtherCAT_Master_BKCUCX.Beckhoff_BKxxxx.Beckhoff_BKxxxxEK1122.A_0019_IL2300_B110_0016.WcState.InputToggle <-> WcState/InputToggle
//     PlcTask Inputs/GVL_iXlinker.EtherCAT_Master_BKCUCX.Beckhoff_BKxxxx.Beckhoff_BKxxxxEK1122.A_0019_IL2300_B110_0016.InfoData.AdsAddr <-> InfoData/AdsAddr
//     PlcTask Inputs/GVL_iXlinker.EtherCAT_Master_BKCUCX.Beckhoff_BKxxxx.Beckhoff_BKxxxxEK1122.A_0019_IL2300_B110_0016.InfoData.AoeNetId <-> InfoData/AoeNetId
//     PlcTask Inputs/GVL_iXlinker.EtherCAT_Master_BKCUCX.Beckhoff_BKxxxx.Beckhoff_BKxxxxEK1122.A_0019_IL2300_B110_0016.InfoData.State <-> InfoData/State
//   PLC/PLC Instance <-> EtherCAT Master BKCUCX/Beckhoff BKxxxx/Beckhoff BKxxxxEK1122/A_0019(IL2300-B110-0016)/Term 19
//     PlcTask Inputs/GVL_iXlinker.EtherCAT_Master_BKCUCX.Beckhoff_BKxxxx.Beckhoff_BKxxxxEK1122.A_0019_IL2300_B110_0016.Term_19.Channel_1.Input <-> Channel 1/Input
//     PlcTask Inputs/GVL_iXlinker.EtherCAT_Master_BKCUCX.Beckhoff_BKxxxx.Beckhoff_BKxxxxEK1122.A_0019_IL2300_B110_0016.Term_19.Channel_2.Input <-> Channel 2/Input
//     PlcTask Inputs/GVL_iXlinker.EtherCAT_Master_BKCUCX.Beckhoff_BKxxxx.Beckhoff_BKxxxxEK1122.A_0019_IL2300_B110_0016.Term_19.Channel_3.Input <-> Channel 3/Input
//     PlcTask Inputs/GVL_iXlinker.EtherCAT_Master_BKCUCX.Beckhoff_BKxxxx.Beckhoff_BKxxxxEK1122.A_0019_IL2300_B110_0016.Term_19.Channel_4.Input <-> Channel 4/Input
//     PlcTask Outputs/GVL_iXlinker.EtherCAT_Master_BKCUCX.Beckhoff_BKxxxx.Beckhoff_BKxxxxEK1122.A_0019_IL2300_B110_0016.Term_19.Channel_1.Output <-> Channel 1/Output
//     PlcTask Outputs/GVL_iXlinker.EtherCAT_Master_BKCUCX.Beckhoff_BKxxxx.Beckhoff_BKxxxxEK1122.A_0019_IL2300_B110_0016.Term_19.Channel_2.Output <-> Channel 2/Output
//     PlcTask Outputs/GVL_iXlinker.EtherCAT_Master_BKCUCX.Beckhoff_BKxxxx.Beckhoff_BKxxxxEK1122.A_0019_IL2300_B110_0016.Term_19.Channel_3.Output <-> Channel 3/Output
//     PlcTask Outputs/GVL_iXlinker.EtherCAT_Master_BKCUCX.Beckhoff_BKxxxx.Beckhoff_BKxxxxEK1122.A_0019_IL2300_B110_0016.Term_19.Channel_4.Output <-> Channel 4/Output
//   PLC/PLC Instance <-> EtherCAT Master BKCUCX/Beckhoff BKxxxx/Beckhoff BKxxxxEK1122/A_0019(IL2300-B110-0016)/Term 390 (Ix1000)
//     PlcTask Inputs/GVL_iXlinker.EtherCAT_Master_BKCUCX.Beckhoff_BKxxxx.Beckhoff_BKxxxxEK1122.A_0019_IL2300_B110_0016.Term_390_Ix1000.Channel_1.Input <-> Channel 1/Input
//     PlcTask Inputs/GVL_iXlinker.EtherCAT_Master_BKCUCX.Beckhoff_BKxxxx.Beckhoff_BKxxxxEK1122.A_0019_IL2300_B110_0016.Term_390_Ix1000.Channel_2.Input <-> Channel 2/Input
//     PlcTask Inputs/GVL_iXlinker.EtherCAT_Master_BKCUCX.Beckhoff_BKxxxx.Beckhoff_BKxxxxEK1122.A_0019_IL2300_B110_0016.Term_390_Ix1000.Channel_3.Input <-> Channel 3/Input
//     PlcTask Inputs/GVL_iXlinker.EtherCAT_Master_BKCUCX.Beckhoff_BKxxxx.Beckhoff_BKxxxxEK1122.A_0019_IL2300_B110_0016.Term_390_Ix1000.Channel_4.Input <-> Channel 4/Input
//     PlcTask Inputs/GVL_iXlinker.EtherCAT_Master_BKCUCX.Beckhoff_BKxxxx.Beckhoff_BKxxxxEK1122.A_0019_IL2300_B110_0016.Term_390_Ix1000.Channel_5.Input <-> Channel 5/Input
//     PlcTask Inputs/GVL_iXlinker.EtherCAT_Master_BKCUCX.Beckhoff_BKxxxx.Beckhoff_BKxxxxEK1122.A_0019_IL2300_B110_0016.Term_390_Ix1000.Channel_6.Input <-> Channel 6/Input
//     PlcTask Inputs/GVL_iXlinker.EtherCAT_Master_BKCUCX.Beckhoff_BKxxxx.Beckhoff_BKxxxxEK1122.A_0019_IL2300_B110_0016.Term_390_Ix1000.Channel_7.Input <-> Channel 7/Input
//     PlcTask Inputs/GVL_iXlinker.EtherCAT_Master_BKCUCX.Beckhoff_BKxxxx.Beckhoff_BKxxxxEK1122.A_0019_IL2300_B110_0016.Term_390_Ix1000.Channel_8.Input <-> Channel 8/Input
//   PLC/PLC Instance <-> EtherCAT Master BKCUCX/Beckhoff BKxxxx/Beckhoff BKxxxxEK1122/A_0020(IL2300-B110-0017)
//     PlcTask Inputs/GVL_iXlinker.EtherCAT_Master_BKCUCX.Beckhoff_BKxxxx.Beckhoff_BKxxxxEK1122.A_0020_IL2300_B110_0017.Inputs.CouplerState <-> Inputs/CouplerState
//     PlcTask Inputs/GVL_iXlinker.EtherCAT_Master_BKCUCX.Beckhoff_BKxxxx.Beckhoff_BKxxxxEK1122.A_0020_IL2300_B110_0017.Outputs.CouplerCtrl <-> Outputs/CouplerCtrl
//     PlcTask Inputs/GVL_iXlinker.EtherCAT_Master_BKCUCX.Beckhoff_BKxxxx.Beckhoff_BKxxxxEK1122.A_0020_IL2300_B110_0017.WcState.WcState <-> WcState/WcState
//     PlcTask Inputs/GVL_iXlinker.EtherCAT_Master_BKCUCX.Beckhoff_BKxxxx.Beckhoff_BKxxxxEK1122.A_0020_IL2300_B110_0017.WcState.InputToggle <-> WcState/InputToggle
//     PlcTask Inputs/GVL_iXlinker.EtherCAT_Master_BKCUCX.Beckhoff_BKxxxx.Beckhoff_BKxxxxEK1122.A_0020_IL2300_B110_0017.InfoData.AdsAddr <-> InfoData/AdsAddr
//     PlcTask Inputs/GVL_iXlinker.EtherCAT_Master_BKCUCX.Beckhoff_BKxxxx.Beckhoff_BKxxxxEK1122.A_0020_IL2300_B110_0017.InfoData.AoeNetId <-> InfoData/AoeNetId
//     PlcTask Inputs/GVL_iXlinker.EtherCAT_Master_BKCUCX.Beckhoff_BKxxxx.Beckhoff_BKxxxxEK1122.A_0020_IL2300_B110_0017.InfoData.State <-> InfoData/State
//   PLC/PLC Instance <-> EtherCAT Master BKCUCX/Beckhoff BKxxxx/Beckhoff BKxxxxEK1122/A_0020(IL2300-B110-0017)/Term 20
//     PlcTask Inputs/GVL_iXlinker.EtherCAT_Master_BKCUCX.Beckhoff_BKxxxx.Beckhoff_BKxxxxEK1122.A_0020_IL2300_B110_0017.Term_20.Channel_1.Input <-> Channel 1/Input
//     PlcTask Inputs/GVL_iXlinker.EtherCAT_Master_BKCUCX.Beckhoff_BKxxxx.Beckhoff_BKxxxxEK1122.A_0020_IL2300_B110_0017.Term_20.Channel_2.Input <-> Channel 2/Input
//     PlcTask Inputs/GVL_iXlinker.EtherCAT_Master_BKCUCX.Beckhoff_BKxxxx.Beckhoff_BKxxxxEK1122.A_0020_IL2300_B110_0017.Term_20.Channel_3.Input <-> Channel 3/Input
//     PlcTask Inputs/GVL_iXlinker.EtherCAT_Master_BKCUCX.Beckhoff_BKxxxx.Beckhoff_BKxxxxEK1122.A_0020_IL2300_B110_0017.Term_20.Channel_4.Input <-> Channel 4/Input
//     PlcTask Outputs/GVL_iXlinker.EtherCAT_Master_BKCUCX.Beckhoff_BKxxxx.Beckhoff_BKxxxxEK1122.A_0020_IL2300_B110_0017.Term_20.Channel_1.Output <-> Channel 1/Output
//     PlcTask Outputs/GVL_iXlinker.EtherCAT_Master_BKCUCX.Beckhoff_BKxxxx.Beckhoff_BKxxxxEK1122.A_0020_IL2300_B110_0017.Term_20.Channel_2.Output <-> Channel 2/Output
//     PlcTask Outputs/GVL_iXlinker.EtherCAT_Master_BKCUCX.Beckhoff_BKxxxx.Beckhoff_BKxxxxEK1122.A_0020_IL2300_B110_0017.Term_20.Channel_3.Output <-> Channel 3/Output
//     PlcTask Outputs/GVL_iXlinker.EtherCAT_Master_BKCUCX.Beckhoff_BKxxxx.Beckhoff_BKxxxxEK1122.A_0020_IL2300_B110_0017.Term_20.Channel_4.Output <-> Channel 4/Output
//   PLC/PLC Instance <-> EtherCAT Master BKCUCX/Beckhoff BKxxxx/Beckhoff BKxxxxEK1122/A_0020(IL2300-B110-0017)/Term 391 (Ix1000)
//     PlcTask Inputs/GVL_iXlinker.EtherCAT_Master_BKCUCX.Beckhoff_BKxxxx.Beckhoff_BKxxxxEK1122.A_0020_IL2300_B110_0017.Term_391_Ix1000.Channel_1.Input <-> Channel 1/Input
//     PlcTask Inputs/GVL_iXlinker.EtherCAT_Master_BKCUCX.Beckhoff_BKxxxx.Beckhoff_BKxxxxEK1122.A_0020_IL2300_B110_0017.Term_391_Ix1000.Channel_2.Input <-> Channel 2/Input
//     PlcTask Inputs/GVL_iXlinker.EtherCAT_Master_BKCUCX.Beckhoff_BKxxxx.Beckhoff_BKxxxxEK1122.A_0020_IL2300_B110_0017.Term_391_Ix1000.Channel_3.Input <-> Channel 3/Input
//     PlcTask Inputs/GVL_iXlinker.EtherCAT_Master_BKCUCX.Beckhoff_BKxxxx.Beckhoff_BKxxxxEK1122.A_0020_IL2300_B110_0017.Term_391_Ix1000.Channel_4.Input <-> Channel 4/Input
//     PlcTask Inputs/GVL_iXlinker.EtherCAT_Master_BKCUCX.Beckhoff_BKxxxx.Beckhoff_BKxxxxEK1122.A_0020_IL2300_B110_0017.Term_391_Ix1000.Channel_5.Input <-> Channel 5/Input
//     PlcTask Inputs/GVL_iXlinker.EtherCAT_Master_BKCUCX.Beckhoff_BKxxxx.Beckhoff_BKxxxxEK1122.A_0020_IL2300_B110_0017.Term_391_Ix1000.Channel_6.Input <-> Channel 6/Input
//     PlcTask Inputs/GVL_iXlinker.EtherCAT_Master_BKCUCX.Beckhoff_BKxxxx.Beckhoff_BKxxxxEK1122.A_0020_IL2300_B110_0017.Term_391_Ix1000.Channel_7.Input <-> Channel 7/Input
//     PlcTask Inputs/GVL_iXlinker.EtherCAT_Master_BKCUCX.Beckhoff_BKxxxx.Beckhoff_BKxxxxEK1122.A_0020_IL2300_B110_0017.Term_391_Ix1000.Channel_8.Input <-> Channel 8/Input
//   PLC/PLC Instance <-> EtherCAT Master BKCUCX/Beckhoff BKxxxx/Beckhoff BKxxxxEK1122/A_0021(IL2301-B110-0016)
//     PlcTask Inputs/GVL_iXlinker.EtherCAT_Master_BKCUCX.Beckhoff_BKxxxx.Beckhoff_BKxxxxEK1122.A_0021_IL2301_B110_0016.Inputs.CouplerState <-> Inputs/CouplerState
//     PlcTask Inputs/GVL_iXlinker.EtherCAT_Master_BKCUCX.Beckhoff_BKxxxx.Beckhoff_BKxxxxEK1122.A_0021_IL2301_B110_0016.Outputs.CouplerCtrl <-> Outputs/CouplerCtrl
//     PlcTask Inputs/GVL_iXlinker.EtherCAT_Master_BKCUCX.Beckhoff_BKxxxx.Beckhoff_BKxxxxEK1122.A_0021_IL2301_B110_0016.WcState.WcState <-> WcState/WcState
//     PlcTask Inputs/GVL_iXlinker.EtherCAT_Master_BKCUCX.Beckhoff_BKxxxx.Beckhoff_BKxxxxEK1122.A_0021_IL2301_B110_0016.WcState.InputToggle <-> WcState/InputToggle
//     PlcTask Inputs/GVL_iXlinker.EtherCAT_Master_BKCUCX.Beckhoff_BKxxxx.Beckhoff_BKxxxxEK1122.A_0021_IL2301_B110_0016.InfoData.AdsAddr <-> InfoData/AdsAddr
//     PlcTask Inputs/GVL_iXlinker.EtherCAT_Master_BKCUCX.Beckhoff_BKxxxx.Beckhoff_BKxxxxEK1122.A_0021_IL2301_B110_0016.InfoData.AoeNetId <-> InfoData/AoeNetId
//     PlcTask Inputs/GVL_iXlinker.EtherCAT_Master_BKCUCX.Beckhoff_BKxxxx.Beckhoff_BKxxxxEK1122.A_0021_IL2301_B110_0016.InfoData.State <-> InfoData/State
//   PLC/PLC Instance <-> EtherCAT Master BKCUCX/Beckhoff BKxxxx/Beckhoff BKxxxxEK1122/A_0021(IL2301-B110-0016)/Term 21
//     PlcTask Inputs/GVL_iXlinker.EtherCAT_Master_BKCUCX.Beckhoff_BKxxxx.Beckhoff_BKxxxxEK1122.A_0021_IL2301_B110_0016.Term_21.Channel_1.Input <-> Channel 1/Input
//     PlcTask Inputs/GVL_iXlinker.EtherCAT_Master_BKCUCX.Beckhoff_BKxxxx.Beckhoff_BKxxxxEK1122.A_0021_IL2301_B110_0016.Term_21.Channel_2.Input <-> Channel 2/Input
//     PlcTask Inputs/GVL_iXlinker.EtherCAT_Master_BKCUCX.Beckhoff_BKxxxx.Beckhoff_BKxxxxEK1122.A_0021_IL2301_B110_0016.Term_21.Channel_3.Input <-> Channel 3/Input
//     PlcTask Inputs/GVL_iXlinker.EtherCAT_Master_BKCUCX.Beckhoff_BKxxxx.Beckhoff_BKxxxxEK1122.A_0021_IL2301_B110_0016.Term_21.Channel_4.Input <-> Channel 4/Input
//     PlcTask Outputs/GVL_iXlinker.EtherCAT_Master_BKCUCX.Beckhoff_BKxxxx.Beckhoff_BKxxxxEK1122.A_0021_IL2301_B110_0016.Term_21.Channel_1.Output <-> Channel 1/Output
//     PlcTask Outputs/GVL_iXlinker.EtherCAT_Master_BKCUCX.Beckhoff_BKxxxx.Beckhoff_BKxxxxEK1122.A_0021_IL2301_B110_0016.Term_21.Channel_2.Output <-> Channel 2/Output
//     PlcTask Outputs/GVL_iXlinker.EtherCAT_Master_BKCUCX.Beckhoff_BKxxxx.Beckhoff_BKxxxxEK1122.A_0021_IL2301_B110_0016.Term_21.Channel_3.Output <-> Channel 3/Output
//     PlcTask Outputs/GVL_iXlinker.EtherCAT_Master_BKCUCX.Beckhoff_BKxxxx.Beckhoff_BKxxxxEK1122.A_0021_IL2301_B110_0016.Term_21.Channel_4.Output <-> Channel 4/Output
//   PLC/PLC Instance <-> EtherCAT Master BKCUCX/Beckhoff BKxxxx/Beckhoff BKxxxxEK1122/A_0021(IL2301-B110-0016)/Term 392 (Ix1000)
//     PlcTask Inputs/GVL_iXlinker.EtherCAT_Master_BKCUCX.Beckhoff_BKxxxx.Beckhoff_BKxxxxEK1122.A_0021_IL2301_B110_0016.Term_392_Ix1000.Channel_1.Input <-> Channel 1/Input
//     PlcTask Inputs/GVL_iXlinker.EtherCAT_Master_BKCUCX.Beckhoff_BKxxxx.Beckhoff_BKxxxxEK1122.A_0021_IL2301_B110_0016.Term_392_Ix1000.Channel_2.Input <-> Channel 2/Input
//     PlcTask Inputs/GVL_iXlinker.EtherCAT_Master_BKCUCX.Beckhoff_BKxxxx.Beckhoff_BKxxxxEK1122.A_0021_IL2301_B110_0016.Term_392_Ix1000.Channel_3.Input <-> Channel 3/Input
//     PlcTask Inputs/GVL_iXlinker.EtherCAT_Master_BKCUCX.Beckhoff_BKxxxx.Beckhoff_BKxxxxEK1122.A_0021_IL2301_B110_0016.Term_392_Ix1000.Channel_4.Input <-> Channel 4/Input
//     PlcTask Inputs/GVL_iXlinker.EtherCAT_Master_BKCUCX.Beckhoff_BKxxxx.Beckhoff_BKxxxxEK1122.A_0021_IL2301_B110_0016.Term_392_Ix1000.Channel_5.Input <-> Channel 5/Input
//     PlcTask Inputs/GVL_iXlinker.EtherCAT_Master_BKCUCX.Beckhoff_BKxxxx.Beckhoff_BKxxxxEK1122.A_0021_IL2301_B110_0016.Term_392_Ix1000.Channel_6.Input <-> Channel 6/Input
//     PlcTask Inputs/GVL_iXlinker.EtherCAT_Master_BKCUCX.Beckhoff_BKxxxx.Beckhoff_BKxxxxEK1122.A_0021_IL2301_B110_0016.Term_392_Ix1000.Channel_7.Input <-> Channel 7/Input
//     PlcTask Inputs/GVL_iXlinker.EtherCAT_Master_BKCUCX.Beckhoff_BKxxxx.Beckhoff_BKxxxxEK1122.A_0021_IL2301_B110_0016.Term_392_Ix1000.Channel_8.Input <-> Channel 8/Input
//   PLC/PLC Instance <-> EtherCAT Master BKCUCX/Beckhoff BKxxxx/Beckhoff BKxxxxEK1122/A_0022(IL2301-B110-0017)
//     PlcTask Inputs/GVL_iXlinker.EtherCAT_Master_BKCUCX.Beckhoff_BKxxxx.Beckhoff_BKxxxxEK1122.A_0022_IL2301_B110_0017.Inputs.CouplerState <-> Inputs/CouplerState
//     PlcTask Inputs/GVL_iXlinker.EtherCAT_Master_BKCUCX.Beckhoff_BKxxxx.Beckhoff_BKxxxxEK1122.A_0022_IL2301_B110_0017.Outputs.CouplerCtrl <-> Outputs/CouplerCtrl
//     PlcTask Inputs/GVL_iXlinker.EtherCAT_Master_BKCUCX.Beckhoff_BKxxxx.Beckhoff_BKxxxxEK1122.A_0022_IL2301_B110_0017.WcState.WcState <-> WcState/WcState
//     PlcTask Inputs/GVL_iXlinker.EtherCAT_Master_BKCUCX.Beckhoff_BKxxxx.Beckhoff_BKxxxxEK1122.A_0022_IL2301_B110_0017.WcState.InputToggle <-> WcState/InputToggle
//     PlcTask Inputs/GVL_iXlinker.EtherCAT_Master_BKCUCX.Beckhoff_BKxxxx.Beckhoff_BKxxxxEK1122.A_0022_IL2301_B110_0017.InfoData.AdsAddr <-> InfoData/AdsAddr
//     PlcTask Inputs/GVL_iXlinker.EtherCAT_Master_BKCUCX.Beckhoff_BKxxxx.Beckhoff_BKxxxxEK1122.A_0022_IL2301_B110_0017.InfoData.AoeNetId <-> InfoData/AoeNetId
//     PlcTask Inputs/GVL_iXlinker.EtherCAT_Master_BKCUCX.Beckhoff_BKxxxx.Beckhoff_BKxxxxEK1122.A_0022_IL2301_B110_0017.InfoData.State <-> InfoData/State
//   PLC/PLC Instance <-> EtherCAT Master BKCUCX/Beckhoff BKxxxx/Beckhoff BKxxxxEK1122/A_0022(IL2301-B110-0017)/Term 22
//     PlcTask Inputs/GVL_iXlinker.EtherCAT_Master_BKCUCX.Beckhoff_BKxxxx.Beckhoff_BKxxxxEK1122.A_0022_IL2301_B110_0017.Term_22.Channel_1.Input <-> Channel 1/Input
//     PlcTask Inputs/GVL_iXlinker.EtherCAT_Master_BKCUCX.Beckhoff_BKxxxx.Beckhoff_BKxxxxEK1122.A_0022_IL2301_B110_0017.Term_22.Channel_2.Input <-> Channel 2/Input
//     PlcTask Inputs/GVL_iXlinker.EtherCAT_Master_BKCUCX.Beckhoff_BKxxxx.Beckhoff_BKxxxxEK1122.A_0022_IL2301_B110_0017.Term_22.Channel_3.Input <-> Channel 3/Input
//     PlcTask Inputs/GVL_iXlinker.EtherCAT_Master_BKCUCX.Beckhoff_BKxxxx.Beckhoff_BKxxxxEK1122.A_0022_IL2301_B110_0017.Term_22.Channel_4.Input <-> Channel 4/Input
//     PlcTask Outputs/GVL_iXlinker.EtherCAT_Master_BKCUCX.Beckhoff_BKxxxx.Beckhoff_BKxxxxEK1122.A_0022_IL2301_B110_0017.Term_22.Channel_1.Output <-> Channel 1/Output
//     PlcTask Outputs/GVL_iXlinker.EtherCAT_Master_BKCUCX.Beckhoff_BKxxxx.Beckhoff_BKxxxxEK1122.A_0022_IL2301_B110_0017.Term_22.Channel_2.Output <-> Channel 2/Output
//     PlcTask Outputs/GVL_iXlinker.EtherCAT_Master_BKCUCX.Beckhoff_BKxxxx.Beckhoff_BKxxxxEK1122.A_0022_IL2301_B110_0017.Term_22.Channel_3.Output <-> Channel 3/Output
//     PlcTask Outputs/GVL_iXlinker.EtherCAT_Master_BKCUCX.Beckhoff_BKxxxx.Beckhoff_BKxxxxEK1122.A_0022_IL2301_B110_0017.Term_22.Channel_4.Output <-> Channel 4/Output
//   PLC/PLC Instance <-> EtherCAT Master BKCUCX/Beckhoff BKxxxx/Beckhoff BKxxxxEK1122/A_0022(IL2301-B110-0017)/Term 393 (Ix1000)
//     PlcTask Inputs/GVL_iXlinker.EtherCAT_Master_BKCUCX.Beckhoff_BKxxxx.Beckhoff_BKxxxxEK1122.A_0022_IL2301_B110_0017.Term_393_Ix1000.Channel_1.Input <-> Channel 1/Input
//     PlcTask Inputs/GVL_iXlinker.EtherCAT_Master_BKCUCX.Beckhoff_BKxxxx.Beckhoff_BKxxxxEK1122.A_0022_IL2301_B110_0017.Term_393_Ix1000.Channel_2.Input <-> Channel 2/Input
//     PlcTask Inputs/GVL_iXlinker.EtherCAT_Master_BKCUCX.Beckhoff_BKxxxx.Beckhoff_BKxxxxEK1122.A_0022_IL2301_B110_0017.Term_393_Ix1000.Channel_3.Input <-> Channel 3/Input
//     PlcTask Inputs/GVL_iXlinker.EtherCAT_Master_BKCUCX.Beckhoff_BKxxxx.Beckhoff_BKxxxxEK1122.A_0022_IL2301_B110_0017.Term_393_Ix1000.Channel_4.Input <-> Channel 4/Input
//     PlcTask Inputs/GVL_iXlinker.EtherCAT_Master_BKCUCX.Beckhoff_BKxxxx.Beckhoff_BKxxxxEK1122.A_0022_IL2301_B110_0017.Term_393_Ix1000.Channel_5.Input <-> Channel 5/Input
//     PlcTask Inputs/GVL_iXlinker.EtherCAT_Master_BKCUCX.Beckhoff_BKxxxx.Beckhoff_BKxxxxEK1122.A_0022_IL2301_B110_0017.Term_393_Ix1000.Channel_6.Input <-> Channel 6/Input
//     PlcTask Inputs/GVL_iXlinker.EtherCAT_Master_BKCUCX.Beckhoff_BKxxxx.Beckhoff_BKxxxxEK1122.A_0022_IL2301_B110_0017.Term_393_Ix1000.Channel_7.Input <-> Channel 7/Input
//     PlcTask Inputs/GVL_iXlinker.EtherCAT_Master_BKCUCX.Beckhoff_BKxxxx.Beckhoff_BKxxxxEK1122.A_0022_IL2301_B110_0017.Term_393_Ix1000.Channel_8.Input <-> Channel 8/Input
//   PLC/PLC Instance <-> EtherCAT Master BKCUCX/Beckhoff BKxxxx/Beckhoff BKxxxxEK1122/A_0023(IL2302-B110-0016)
//     PlcTask Inputs/GVL_iXlinker.EtherCAT_Master_BKCUCX.Beckhoff_BKxxxx.Beckhoff_BKxxxxEK1122.A_0023_IL2302_B110_0016.Inputs.CouplerState <-> Inputs/CouplerState
//     PlcTask Inputs/GVL_iXlinker.EtherCAT_Master_BKCUCX.Beckhoff_BKxxxx.Beckhoff_BKxxxxEK1122.A_0023_IL2302_B110_0016.Outputs.CouplerCtrl <-> Outputs/CouplerCtrl
//     PlcTask Inputs/GVL_iXlinker.EtherCAT_Master_BKCUCX.Beckhoff_BKxxxx.Beckhoff_BKxxxxEK1122.A_0023_IL2302_B110_0016.WcState.WcState <-> WcState/WcState
//     PlcTask Inputs/GVL_iXlinker.EtherCAT_Master_BKCUCX.Beckhoff_BKxxxx.Beckhoff_BKxxxxEK1122.A_0023_IL2302_B110_0016.WcState.InputToggle <-> WcState/InputToggle
//     PlcTask Inputs/GVL_iXlinker.EtherCAT_Master_BKCUCX.Beckhoff_BKxxxx.Beckhoff_BKxxxxEK1122.A_0023_IL2302_B110_0016.InfoData.AdsAddr <-> InfoData/AdsAddr
//     PlcTask Inputs/GVL_iXlinker.EtherCAT_Master_BKCUCX.Beckhoff_BKxxxx.Beckhoff_BKxxxxEK1122.A_0023_IL2302_B110_0016.InfoData.AoeNetId <-> InfoData/AoeNetId
//     PlcTask Inputs/GVL_iXlinker.EtherCAT_Master_BKCUCX.Beckhoff_BKxxxx.Beckhoff_BKxxxxEK1122.A_0023_IL2302_B110_0016.InfoData.State <-> InfoData/State
//   PLC/PLC Instance <-> EtherCAT Master BKCUCX/Beckhoff BKxxxx/Beckhoff BKxxxxEK1122/A_0023(IL2302-B110-0016)/Term 23
//     PlcTask Inputs/GVL_iXlinker.EtherCAT_Master_BKCUCX.Beckhoff_BKxxxx.Beckhoff_BKxxxxEK1122.A_0023_IL2302_B110_0016.Term_23.Channel_1.Input <-> Channel 1/Input
//     PlcTask Inputs/GVL_iXlinker.EtherCAT_Master_BKCUCX.Beckhoff_BKxxxx.Beckhoff_BKxxxxEK1122.A_0023_IL2302_B110_0016.Term_23.Channel_2.Input <-> Channel 2/Input
//     PlcTask Inputs/GVL_iXlinker.EtherCAT_Master_BKCUCX.Beckhoff_BKxxxx.Beckhoff_BKxxxxEK1122.A_0023_IL2302_B110_0016.Term_23.Channel_3.Input <-> Channel 3/Input
//     PlcTask Inputs/GVL_iXlinker.EtherCAT_Master_BKCUCX.Beckhoff_BKxxxx.Beckhoff_BKxxxxEK1122.A_0023_IL2302_B110_0016.Term_23.Channel_4.Input <-> Channel 4/Input
//     PlcTask Outputs/GVL_iXlinker.EtherCAT_Master_BKCUCX.Beckhoff_BKxxxx.Beckhoff_BKxxxxEK1122.A_0023_IL2302_B110_0016.Term_23.Channel_1.Output <-> Channel 1/Output
//     PlcTask Outputs/GVL_iXlinker.EtherCAT_Master_BKCUCX.Beckhoff_BKxxxx.Beckhoff_BKxxxxEK1122.A_0023_IL2302_B110_0016.Term_23.Channel_2.Output <-> Channel 2/Output
//     PlcTask Outputs/GVL_iXlinker.EtherCAT_Master_BKCUCX.Beckhoff_BKxxxx.Beckhoff_BKxxxxEK1122.A_0023_IL2302_B110_0016.Term_23.Channel_3.Output <-> Channel 3/Output
//     PlcTask Outputs/GVL_iXlinker.EtherCAT_Master_BKCUCX.Beckhoff_BKxxxx.Beckhoff_BKxxxxEK1122.A_0023_IL2302_B110_0016.Term_23.Channel_4.Output <-> Channel 4/Output
//   PLC/PLC Instance <-> EtherCAT Master BKCUCX/Beckhoff BKxxxx/Beckhoff BKxxxxEK1122/A_0023(IL2302-B110-0016)/Term 394 (Ix1000)
//     PlcTask Inputs/GVL_iXlinker.EtherCAT_Master_BKCUCX.Beckhoff_BKxxxx.Beckhoff_BKxxxxEK1122.A_0023_IL2302_B110_0016.Term_394_Ix1000.Channel_1.Input <-> Channel 1/Input
//     PlcTask Inputs/GVL_iXlinker.EtherCAT_Master_BKCUCX.Beckhoff_BKxxxx.Beckhoff_BKxxxxEK1122.A_0023_IL2302_B110_0016.Term_394_Ix1000.Channel_2.Input <-> Channel 2/Input
//     PlcTask Inputs/GVL_iXlinker.EtherCAT_Master_BKCUCX.Beckhoff_BKxxxx.Beckhoff_BKxxxxEK1122.A_0023_IL2302_B110_0016.Term_394_Ix1000.Channel_3.Input <-> Channel 3/Input
//     PlcTask Inputs/GVL_iXlinker.EtherCAT_Master_BKCUCX.Beckhoff_BKxxxx.Beckhoff_BKxxxxEK1122.A_0023_IL2302_B110_0016.Term_394_Ix1000.Channel_4.Input <-> Channel 4/Input
//     PlcTask Inputs/GVL_iXlinker.EtherCAT_Master_BKCUCX.Beckhoff_BKxxxx.Beckhoff_BKxxxxEK1122.A_0023_IL2302_B110_0016.Term_394_Ix1000.Channel_5.Input <-> Channel 5/Input
//     PlcTask Inputs/GVL_iXlinker.EtherCAT_Master_BKCUCX.Beckhoff_BKxxxx.Beckhoff_BKxxxxEK1122.A_0023_IL2302_B110_0016.Term_394_Ix1000.Channel_6.Input <-> Channel 6/Input
//     PlcTask Inputs/GVL_iXlinker.EtherCAT_Master_BKCUCX.Beckhoff_BKxxxx.Beckhoff_BKxxxxEK1122.A_0023_IL2302_B110_0016.Term_394_Ix1000.Channel_7.Input <-> Channel 7/Input
//     PlcTask Inputs/GVL_iXlinker.EtherCAT_Master_BKCUCX.Beckhoff_BKxxxx.Beckhoff_BKxxxxEK1122.A_0023_IL2302_B110_0016.Term_394_Ix1000.Channel_8.Input <-> Channel 8/Input
//   PLC/PLC Instance <-> EtherCAT Master BKCUCX/Beckhoff BKxxxx/Beckhoff BKxxxxEK1122/A_0024(IL2302-B110-0017)
//     PlcTask Inputs/GVL_iXlinker.EtherCAT_Master_BKCUCX.Beckhoff_BKxxxx.Beckhoff_BKxxxxEK1122.A_0024_IL2302_B110_0017.Inputs.CouplerState <-> Inputs/CouplerState
//     PlcTask Inputs/GVL_iXlinker.EtherCAT_Master_BKCUCX.Beckhoff_BKxxxx.Beckhoff_BKxxxxEK1122.A_0024_IL2302_B110_0017.Outputs.CouplerCtrl <-> Outputs/CouplerCtrl
//     PlcTask Inputs/GVL_iXlinker.EtherCAT_Master_BKCUCX.Beckhoff_BKxxxx.Beckhoff_BKxxxxEK1122.A_0024_IL2302_B110_0017.WcState.WcState <-> WcState/WcState
//     PlcTask Inputs/GVL_iXlinker.EtherCAT_Master_BKCUCX.Beckhoff_BKxxxx.Beckhoff_BKxxxxEK1122.A_0024_IL2302_B110_0017.WcState.InputToggle <-> WcState/InputToggle
//     PlcTask Inputs/GVL_iXlinker.EtherCAT_Master_BKCUCX.Beckhoff_BKxxxx.Beckhoff_BKxxxxEK1122.A_0024_IL2302_B110_0017.InfoData.AdsAddr <-> InfoData/AdsAddr
//     PlcTask Inputs/GVL_iXlinker.EtherCAT_Master_BKCUCX.Beckhoff_BKxxxx.Beckhoff_BKxxxxEK1122.A_0024_IL2302_B110_0017.InfoData.AoeNetId <-> InfoData/AoeNetId
//     PlcTask Inputs/GVL_iXlinker.EtherCAT_Master_BKCUCX.Beckhoff_BKxxxx.Beckhoff_BKxxxxEK1122.A_0024_IL2302_B110_0017.InfoData.State <-> InfoData/State
//   PLC/PLC Instance <-> EtherCAT Master BKCUCX/Beckhoff BKxxxx/Beckhoff BKxxxxEK1122/A_0024(IL2302-B110-0017)/Term 24
//     PlcTask Inputs/GVL_iXlinker.EtherCAT_Master_BKCUCX.Beckhoff_BKxxxx.Beckhoff_BKxxxxEK1122.A_0024_IL2302_B110_0017.Term_24.Channel_1.Input <-> Channel 1/Input
//     PlcTask Inputs/GVL_iXlinker.EtherCAT_Master_BKCUCX.Beckhoff_BKxxxx.Beckhoff_BKxxxxEK1122.A_0024_IL2302_B110_0017.Term_24.Channel_2.Input <-> Channel 2/Input
//     PlcTask Inputs/GVL_iXlinker.EtherCAT_Master_BKCUCX.Beckhoff_BKxxxx.Beckhoff_BKxxxxEK1122.A_0024_IL2302_B110_0017.Term_24.Channel_3.Input <-> Channel 3/Input
//     PlcTask Inputs/GVL_iXlinker.EtherCAT_Master_BKCUCX.Beckhoff_BKxxxx.Beckhoff_BKxxxxEK1122.A_0024_IL2302_B110_0017.Term_24.Channel_4.Input <-> Channel 4/Input
//     PlcTask Outputs/GVL_iXlinker.EtherCAT_Master_BKCUCX.Beckhoff_BKxxxx.Beckhoff_BKxxxxEK1122.A_0024_IL2302_B110_0017.Term_24.Channel_1.Output <-> Channel 1/Output
//     PlcTask Outputs/GVL_iXlinker.EtherCAT_Master_BKCUCX.Beckhoff_BKxxxx.Beckhoff_BKxxxxEK1122.A_0024_IL2302_B110_0017.Term_24.Channel_2.Output <-> Channel 2/Output
//     PlcTask Outputs/GVL_iXlinker.EtherCAT_Master_BKCUCX.Beckhoff_BKxxxx.Beckhoff_BKxxxxEK1122.A_0024_IL2302_B110_0017.Term_24.Channel_3.Output <-> Channel 3/Output
//     PlcTask Outputs/GVL_iXlinker.EtherCAT_Master_BKCUCX.Beckhoff_BKxxxx.Beckhoff_BKxxxxEK1122.A_0024_IL2302_B110_0017.Term_24.Channel_4.Output <-> Channel 4/Output
//   PLC/PLC Instance <-> EtherCAT Master BKCUCX/Beckhoff BKxxxx/Beckhoff BKxxxxEK1122/A_0024(IL2302-B110-0017)/Term 395 (Ix1000)
//     PlcTask Inputs/GVL_iXlinker.EtherCAT_Master_BKCUCX.Beckhoff_BKxxxx.Beckhoff_BKxxxxEK1122.A_0024_IL2302_B110_0017.Term_395_Ix1000.Channel_1.Input <-> Channel 1/Input
//     PlcTask Inputs/GVL_iXlinker.EtherCAT_Master_BKCUCX.Beckhoff_BKxxxx.Beckhoff_BKxxxxEK1122.A_0024_IL2302_B110_0017.Term_395_Ix1000.Channel_2.Input <-> Channel 2/Input
//     PlcTask Inputs/GVL_iXlinker.EtherCAT_Master_BKCUCX.Beckhoff_BKxxxx.Beckhoff_BKxxxxEK1122.A_0024_IL2302_B110_0017.Term_395_Ix1000.Channel_3.Input <-> Channel 3/Input
//     PlcTask Inputs/GVL_iXlinker.EtherCAT_Master_BKCUCX.Beckhoff_BKxxxx.Beckhoff_BKxxxxEK1122.A_0024_IL2302_B110_0017.Term_395_Ix1000.Channel_4.Input <-> Channel 4/Input
//     PlcTask Inputs/GVL_iXlinker.EtherCAT_Master_BKCUCX.Beckhoff_BKxxxx.Beckhoff_BKxxxxEK1122.A_0024_IL2302_B110_0017.Term_395_Ix1000.Channel_5.Input <-> Channel 5/Input
//     PlcTask Inputs/GVL_iXlinker.EtherCAT_Master_BKCUCX.Beckhoff_BKxxxx.Beckhoff_BKxxxxEK1122.A_0024_IL2302_B110_0017.Term_395_Ix1000.Channel_6.Input <-> Channel 6/Input
//     PlcTask Inputs/GVL_iXlinker.EtherCAT_Master_BKCUCX.Beckhoff_BKxxxx.Beckhoff_BKxxxxEK1122.A_0024_IL2302_B110_0017.Term_395_Ix1000.Channel_7.Input <-> Channel 7/Input
//     PlcTask Inputs/GVL_iXlinker.EtherCAT_Master_BKCUCX.Beckhoff_BKxxxx.Beckhoff_BKxxxxEK1122.A_0024_IL2302_B110_0017.Term_395_Ix1000.Channel_8.Input <-> Channel 8/Input
//   PLC/PLC Instance <-> EtherCAT Master BKCUCX/Beckhoff BKxxxx/A_0015(BK1250-0000-0016)
//     PlcTask Inputs/GVL_iXlinker.EtherCAT_Master_BKCUCX.Beckhoff_BKxxxx.A_0015_BK1250_0000_0016.Inputs.CouplerState <-> Inputs/CouplerState
//     PlcTask Inputs/GVL_iXlinker.EtherCAT_Master_BKCUCX.Beckhoff_BKxxxx.A_0015_BK1250_0000_0016.Outputs.CouplerCtrl <-> Outputs/CouplerCtrl
//     PlcTask Inputs/GVL_iXlinker.EtherCAT_Master_BKCUCX.Beckhoff_BKxxxx.A_0015_BK1250_0000_0016.WcState.WcState <-> WcState/WcState
//     PlcTask Inputs/GVL_iXlinker.EtherCAT_Master_BKCUCX.Beckhoff_BKxxxx.A_0015_BK1250_0000_0016.WcState.InputToggle <-> WcState/InputToggle
//     PlcTask Inputs/GVL_iXlinker.EtherCAT_Master_BKCUCX.Beckhoff_BKxxxx.A_0015_BK1250_0000_0016.InfoData.AdsAddr <-> InfoData/AdsAddr
//     PlcTask Inputs/GVL_iXlinker.EtherCAT_Master_BKCUCX.Beckhoff_BKxxxx.A_0015_BK1250_0000_0016.InfoData.AoeNetId <-> InfoData/AoeNetId
//     PlcTask Inputs/GVL_iXlinker.EtherCAT_Master_BKCUCX.Beckhoff_BKxxxx.A_0015_BK1250_0000_0016.InfoData.State <-> InfoData/State
//   PLC/PLC Instance <-> EtherCAT Master BKCUCX/Beckhoff BKxxxx/A_0015(BK1250-0000-0016)/Term 396 (KL1002)
//     PlcTask Inputs/GVL_iXlinker.EtherCAT_Master_BKCUCX.Beckhoff_BKxxxx.A_0015_BK1250_0000_0016.Term_396_KL1002.Channel_1.Input <-> Channel 1/Input
//     PlcTask Inputs/GVL_iXlinker.EtherCAT_Master_BKCUCX.Beckhoff_BKxxxx.A_0015_BK1250_0000_0016.Term_396_KL1002.Channel_2.Input <-> Channel 2/Input
//   PLC/PLC Instance <-> EtherCAT Master BKCUCX/Beckhoff CUxxxx
//     PlcTask Inputs/GVL_iXlinker.EtherCAT_Master_BKCUCX.Beckhoff_CUxxxx.InfoData.State <-> InfoData/State
//   PLC/PLC Instance <-> EtherCAT Master BKCUCX/Beckhoff CUxxxx/Beckhoff CUxxxxEK1122
//     PlcTask Inputs/GVL_iXlinker.EtherCAT_Master_BKCUCX.Beckhoff_CUxxxx.Beckhoff_CUxxxxEK1122.InfoData.State <-> InfoData/State
//   PLC/PLC Instance <-> EtherCAT Master BKCUCX/Beckhoff CUxxxx/Beckhoff CUxxxxEK1122/Beckhoff CUxxxxsub EK1100
//     PlcTask Inputs/GVL_iXlinker.EtherCAT_Master_BKCUCX.Beckhoff_CUxxxx.Beckhoff_CUxxxxEK1122.Beckhoff_CUxxxxsub_EK1100.InfoData.State <-> InfoData/State
//   PLC/PLC Instance <-> EtherCAT Master BKCUCX/Beckhoff CUxxxx/Beckhoff CUxxxxEK1122/A_0001(CU1123-0000-0016)
//     PlcTask Inputs/GVL_iXlinker.EtherCAT_Master_BKCUCX.Beckhoff_CUxxxx.Beckhoff_CUxxxxEK1122.A_0001_CU1123_0000_0016.InfoData.State <-> InfoData/State
//   PLC/PLC Instance <-> EtherCAT Master BKCUCX/Beckhoff CUxxxx/Beckhoff CUxxxxEK1122/A_0001(CU1123-0000-0016)/A_0002(CU1123-0010-0016)
//     PlcTask Inputs/GVL_iXlinker.EtherCAT_Master_BKCUCX.Beckhoff_CUxxxx.Beckhoff_CUxxxxEK1122.A_0001_CU1123_0000_0016.A_0002_CU1123_0010_0016.InfoData.State <-> InfoData/State
//   PLC/PLC Instance <-> EtherCAT Master BKCUCX/Beckhoff CUxxxx/Beckhoff CUxxxxEK1122/A_0001(CU1123-0000-0016)/A_0002(CU1123-0010-0016)/A_0003(CU1124-0000-0016)
//     PlcTask Inputs/GVL_iXlinker.EtherCAT_Master_BKCUCX.Beckhoff_CUxxxx.Beckhoff_CUxxxxEK1122.A_0001_CU1123_0000_0016.A_0002_CU1123_0010_0016.A_0003_CU1124_0000_0016.InfoData.State <-> InfoData/State
//   PLC/PLC Instance <-> EtherCAT Master BKCUCX/Beckhoff CUxxxx/Beckhoff CUxxxxEK1122/A_0001(CU1123-0000-0016)/A_0002(CU1123-0010-0016)/A_0003(CU1124-0000-0016)/A_0004(CU1128-0000-0000)
//     PlcTask Inputs/GVL_iXlinker.EtherCAT_Master_BKCUCX.Beckhoff_CUxxxx.Beckhoff_CUxxxxEK1122.A_0001_CU1123_0000_0016.A_0002_CU1123_0010_0016.A_0003_CU1124_0000_0016.A_0004_CU1128_0000_0000.InfoData.State <-> InfoData/State
//   PLC/PLC Instance <-> EtherCAT Master BKCUCX/Beckhoff CUxxxx/Beckhoff CUxxxxEK1122/A_0001(CU1123-0000-0016)/A_0002(CU1123-0010-0016)/A_0003(CU1124-0000-0016)/A_0004(CU1128-0000-0000)/A_0005(CU1128-0000-0001)
//     PlcTask Inputs/GVL_iXlinker.EtherCAT_Master_BKCUCX.Beckhoff_CUxxxx.Beckhoff_CUxxxxEK1122.A_0001_CU1123_0000_0016.A_0002_CU1123_0010_0016.A_0003_CU1124_0000_0016.A_0004_CU1128_0000_0000.A_0005_CU1128_0000_0001.InfoData.State <-> InfoData/State
//   PLC/PLC Instance <-> EtherCAT Master BKCUCX/Beckhoff CUxxxx/Beckhoff CUxxxxEK1122/A_0001(CU1123-0000-0016)/A_0002(CU1123-0010-0016)/A_0003(CU1124-0000-0016)/A_0004(CU1128-0000-0000)/A_0005(CU1128-0000-0001)/A_0006(CU1128-0000-0002)
//     PlcTask Inputs/GVL_iXlinker.EtherCAT_Master_BKCUCX.Beckhoff_CUxxxx.Beckhoff_CUxxxxEK1122.A_0001_CU1123_0000_0016.A_0002_CU1123_0010_0016.A_0003_CU1124_0000_0016.A_0004_CU1128_0000_0000.A_0005_CU1128_0000_0001.A_0006_CU1128_0000_0002.InfoData.State <-> InfoData/State
//   PLC/PLC Instance <-> EtherCAT Master BKCUCX/Beckhoff CUxxxx/Beckhoff CUxxxxEK1122/A_0001(CU1123-0000-0016)/A_0002(CU1123-0010-0016)/A_0003(CU1124-0000-0016)/A_0004(CU1128-0000-0000)/A_0005(CU1128-0000-0001)/A_0006(CU1128-0000-0002)/A_0007(CU1521-0010-0000)
//     PlcTask Inputs/GVL_iXlinker.EtherCAT_Master_BKCUCX.Beckhoff_CUxxxx.Beckhoff_CUxxxxEK1122.A_0001_CU1123_0000_0016.A_0002_CU1123_0010_0016.A_0003_CU1124_0000_0016.A_0004_CU1128_0000_0000.A_0005_CU1128_0000_0001.A_0006_CU1128_0000_0002.A_0007_CU1521_0010_0000.InfoData.State <-> InfoData/State
//   PLC/PLC Instance <-> EtherCAT Master BKCUCX/Beckhoff CUxxxx/Beckhoff CUxxxxEK1122/A_0001(CU1123-0000-0016)/A_0002(CU1123-0010-0016)/A_0003(CU1124-0000-0016)/A_0004(CU1128-0000-0000)/A_0005(CU1128-0000-0001)/A_0006(CU1128-0000-0002)/A_0008(CU1561-0000-0000)
//     PlcTask Inputs/GVL_iXlinker.EtherCAT_Master_BKCUCX.Beckhoff_CUxxxx.Beckhoff_CUxxxxEK1122.A_0001_CU1123_0000_0016.A_0002_CU1123_0010_0016.A_0003_CU1124_0000_0016.A_0004_CU1128_0000_0000.A_0005_CU1128_0000_0001.A_0006_CU1128_0000_0002.A_0008_CU1561_0000_0000.InfoData.State <-> InfoData/State
//   PLC/PLC Instance <-> EtherCAT Master BKCUCX/Beckhoff CUxxxx/Beckhoff CUxxxxEK1122/A_0001(CU1123-0000-0016)/A_0002(CU1123-0010-0016)/A_0003(CU1124-0000-0016)/A_0004(CU1128-0000-0000)/A_0005(CU1128-0000-0001)/A_0006(CU1128-0000-0002)/A_0009(CU2508-0000-0000)
//     PlcTask Inputs/GVL_iXlinker.EtherCAT_Master_BKCUCX.Beckhoff_CUxxxx.Beckhoff_CUxxxxEK1122.A_0001_CU1123_0000_0016.A_0002_CU1123_0010_0016.A_0003_CU1124_0000_0016.A_0004_CU1128_0000_0000.A_0005_CU1128_0000_0001.A_0006_CU1128_0000_0002.A_0009_CU2508_0000_0000.InfoData.State <-> InfoData/State
//   PLC/PLC Instance <-> EtherCAT Master BKCUCX/Beckhoff CUxxxx/Beckhoff CUxxxxEK1122/A_0001(CU1123-0000-0016)/A_0002(CU1123-0010-0016)/A_0003(CU1124-0000-0016)/A_0004(CU1128-0000-0000)/A_0005(CU1128-0000-0001)/A_0006(CU1128-0000-0002)/A_0010(CU2508-0000-0016)
//     PlcTask Inputs/GVL_iXlinker.EtherCAT_Master_BKCUCX.Beckhoff_CUxxxx.Beckhoff_CUxxxxEK1122.A_0001_CU1123_0000_0016.A_0002_CU1123_0010_0016.A_0003_CU1124_0000_0016.A_0004_CU1128_0000_0000.A_0005_CU1128_0000_0001.A_0006_CU1128_0000_0002.A_0010_CU2508_0000_0016.InfoData.AdsAddr <-> InfoData/AdsAddr
//     PlcTask Inputs/GVL_iXlinker.EtherCAT_Master_BKCUCX.Beckhoff_CUxxxx.Beckhoff_CUxxxxEK1122.A_0001_CU1123_0000_0016.A_0002_CU1123_0010_0016.A_0003_CU1124_0000_0016.A_0004_CU1128_0000_0000.A_0005_CU1128_0000_0001.A_0006_CU1128_0000_0002.A_0010_CU2508_0000_0016.InfoData.State <-> InfoData/State
//   PLC/PLC Instance <-> EtherCAT Master BKCUCX/Beckhoff CUxxxx/Beckhoff CUxxxxEK1122/A_0001(CU1123-0000-0016)/A_0002(CU1123-0010-0016)/A_0003(CU1124-0000-0016)/A_0004(CU1128-0000-0000)/A_0005(CU1128-0000-0001)/A_0006(CU1128-0000-0002)/A_0011(CU2508-0000-0017)
//     PlcTask Inputs/GVL_iXlinker.EtherCAT_Master_BKCUCX.Beckhoff_CUxxxx.Beckhoff_CUxxxxEK1122.A_0001_CU1123_0000_0016.A_0002_CU1123_0010_0016.A_0003_CU1124_0000_0016.A_0004_CU1128_0000_0000.A_0005_CU1128_0000_0001.A_0006_CU1128_0000_0002.A_0011_CU2508_0000_0017.EPM_Inputs_Channel_1.Dropped_frames_rx <-> EPM Inputs Channel 1/Dropped frames rx
//     PlcTask Inputs/GVL_iXlinker.EtherCAT_Master_BKCUCX.Beckhoff_CUxxxx.Beckhoff_CUxxxxEK1122.A_0001_CU1123_0000_0016.A_0002_CU1123_0010_0016.A_0003_CU1124_0000_0016.A_0004_CU1128_0000_0000.A_0005_CU1128_0000_0001.A_0006_CU1128_0000_0002.A_0011_CU2508_0000_0017.EPM_Inputs_Channel_2.Dropped_frames_rx <-> EPM Inputs Channel 2/Dropped frames rx
//     PlcTask Inputs/GVL_iXlinker.EtherCAT_Master_BKCUCX.Beckhoff_CUxxxx.Beckhoff_CUxxxxEK1122.A_0001_CU1123_0000_0016.A_0002_CU1123_0010_0016.A_0003_CU1124_0000_0016.A_0004_CU1128_0000_0000.A_0005_CU1128_0000_0001.A_0006_CU1128_0000_0002.A_0011_CU2508_0000_0017.EPM_Inputs_Channel_3.Dropped_frames_rx <-> EPM Inputs Channel 3/Dropped frames rx
//     PlcTask Inputs/GVL_iXlinker.EtherCAT_Master_BKCUCX.Beckhoff_CUxxxx.Beckhoff_CUxxxxEK1122.A_0001_CU1123_0000_0016.A_0002_CU1123_0010_0016.A_0003_CU1124_0000_0016.A_0004_CU1128_0000_0000.A_0005_CU1128_0000_0001.A_0006_CU1128_0000_0002.A_0011_CU2508_0000_0017.EPM_Inputs_Channel_4.Dropped_frames_rx <-> EPM Inputs Channel 4/Dropped frames rx
//     PlcTask Inputs/GVL_iXlinker.EtherCAT_Master_BKCUCX.Beckhoff_CUxxxx.Beckhoff_CUxxxxEK1122.A_0001_CU1123_0000_0016.A_0002_CU1123_0010_0016.A_0003_CU1124_0000_0016.A_0004_CU1128_0000_0000.A_0005_CU1128_0000_0001.A_0006_CU1128_0000_0002.A_0011_CU2508_0000_0017.EPM_Inputs_Channel_5.Dropped_frames_rx <-> EPM Inputs Channel 5/Dropped frames rx
//     PlcTask Inputs/GVL_iXlinker.EtherCAT_Master_BKCUCX.Beckhoff_CUxxxx.Beckhoff_CUxxxxEK1122.A_0001_CU1123_0000_0016.A_0002_CU1123_0010_0016.A_0003_CU1124_0000_0016.A_0004_CU1128_0000_0000.A_0005_CU1128_0000_0001.A_0006_CU1128_0000_0002.A_0011_CU2508_0000_0017.EPM_Inputs_Channel_6.Dropped_frames_rx <-> EPM Inputs Channel 6/Dropped frames rx
//     PlcTask Inputs/GVL_iXlinker.EtherCAT_Master_BKCUCX.Beckhoff_CUxxxx.Beckhoff_CUxxxxEK1122.A_0001_CU1123_0000_0016.A_0002_CU1123_0010_0016.A_0003_CU1124_0000_0016.A_0004_CU1128_0000_0000.A_0005_CU1128_0000_0001.A_0006_CU1128_0000_0002.A_0011_CU2508_0000_0017.EPM_Inputs_Channel_7.Dropped_frames_rx <-> EPM Inputs Channel 7/Dropped frames rx
//     PlcTask Inputs/GVL_iXlinker.EtherCAT_Master_BKCUCX.Beckhoff_CUxxxx.Beckhoff_CUxxxxEK1122.A_0001_CU1123_0000_0016.A_0002_CU1123_0010_0016.A_0003_CU1124_0000_0016.A_0004_CU1128_0000_0000.A_0005_CU1128_0000_0001.A_0006_CU1128_0000_0002.A_0011_CU2508_0000_0017.EPM_Inputs_Channel_8.Dropped_frames_rx <-> EPM Inputs Channel 8/Dropped frames rx
//     PlcTask Inputs/GVL_iXlinker.EtherCAT_Master_BKCUCX.Beckhoff_CUxxxx.Beckhoff_CUxxxxEK1122.A_0001_CU1123_0000_0016.A_0002_CU1123_0010_0016.A_0003_CU1124_0000_0016.A_0004_CU1128_0000_0000.A_0005_CU1128_0000_0001.A_0006_CU1128_0000_0002.A_0011_CU2508_0000_0017.EPM_Inputs_Channel_9.Dropped_frames_rx <-> EPM Inputs Channel 9/Dropped frames rx
//     PlcTask Inputs/GVL_iXlinker.EtherCAT_Master_BKCUCX.Beckhoff_CUxxxx.Beckhoff_CUxxxxEK1122.A_0001_CU1123_0000_0016.A_0002_CU1123_0010_0016.A_0003_CU1124_0000_0016.A_0004_CU1128_0000_0000.A_0005_CU1128_0000_0001.A_0006_CU1128_0000_0002.A_0011_CU2508_0000_0017.EPM_Inputs_Channel_10.Dropped_frames_rx <-> EPM Inputs Channel 10/Dropped frames rx
//     PlcTask Inputs/GVL_iXlinker.EtherCAT_Master_BKCUCX.Beckhoff_CUxxxx.Beckhoff_CUxxxxEK1122.A_0001_CU1123_0000_0016.A_0002_CU1123_0010_0016.A_0003_CU1124_0000_0016.A_0004_CU1128_0000_0000.A_0005_CU1128_0000_0001.A_0006_CU1128_0000_0002.A_0011_CU2508_0000_0017.EPM_Inputs_Channel_1.Dropped_frames_tx <-> EPM Inputs Channel 1/Dropped frames tx
//     PlcTask Inputs/GVL_iXlinker.EtherCAT_Master_BKCUCX.Beckhoff_CUxxxx.Beckhoff_CUxxxxEK1122.A_0001_CU1123_0000_0016.A_0002_CU1123_0010_0016.A_0003_CU1124_0000_0016.A_0004_CU1128_0000_0000.A_0005_CU1128_0000_0001.A_0006_CU1128_0000_0002.A_0011_CU2508_0000_0017.EPM_Inputs_Channel_2.Dropped_frames_tx <-> EPM Inputs Channel 2/Dropped frames tx
//     PlcTask Inputs/GVL_iXlinker.EtherCAT_Master_BKCUCX.Beckhoff_CUxxxx.Beckhoff_CUxxxxEK1122.A_0001_CU1123_0000_0016.A_0002_CU1123_0010_0016.A_0003_CU1124_0000_0016.A_0004_CU1128_0000_0000.A_0005_CU1128_0000_0001.A_0006_CU1128_0000_0002.A_0011_CU2508_0000_0017.EPM_Inputs_Channel_3.Dropped_frames_tx <-> EPM Inputs Channel 3/Dropped frames tx
//     PlcTask Inputs/GVL_iXlinker.EtherCAT_Master_BKCUCX.Beckhoff_CUxxxx.Beckhoff_CUxxxxEK1122.A_0001_CU1123_0000_0016.A_0002_CU1123_0010_0016.A_0003_CU1124_0000_0016.A_0004_CU1128_0000_0000.A_0005_CU1128_0000_0001.A_0006_CU1128_0000_0002.A_0011_CU2508_0000_0017.EPM_Inputs_Channel_4.Dropped_frames_tx <-> EPM Inputs Channel 4/Dropped frames tx
//     PlcTask Inputs/GVL_iXlinker.EtherCAT_Master_BKCUCX.Beckhoff_CUxxxx.Beckhoff_CUxxxxEK1122.A_0001_CU1123_0000_0016.A_0002_CU1123_0010_0016.A_0003_CU1124_0000_0016.A_0004_CU1128_0000_0000.A_0005_CU1128_0000_0001.A_0006_CU1128_0000_0002.A_0011_CU2508_0000_0017.EPM_Inputs_Channel_5.Dropped_frames_tx <-> EPM Inputs Channel 5/Dropped frames tx
//     PlcTask Inputs/GVL_iXlinker.EtherCAT_Master_BKCUCX.Beckhoff_CUxxxx.Beckhoff_CUxxxxEK1122.A_0001_CU1123_0000_0016.A_0002_CU1123_0010_0016.A_0003_CU1124_0000_0016.A_0004_CU1128_0000_0000.A_0005_CU1128_0000_0001.A_0006_CU1128_0000_0002.A_0011_CU2508_0000_0017.EPM_Inputs_Channel_6.Dropped_frames_tx <-> EPM Inputs Channel 6/Dropped frames tx
//     PlcTask Inputs/GVL_iXlinker.EtherCAT_Master_BKCUCX.Beckhoff_CUxxxx.Beckhoff_CUxxxxEK1122.A_0001_CU1123_0000_0016.A_0002_CU1123_0010_0016.A_0003_CU1124_0000_0016.A_0004_CU1128_0000_0000.A_0005_CU1128_0000_0001.A_0006_CU1128_0000_0002.A_0011_CU2508_0000_0017.EPM_Inputs_Channel_7.Dropped_frames_tx <-> EPM Inputs Channel 7/Dropped frames tx
//     PlcTask Inputs/GVL_iXlinker.EtherCAT_Master_BKCUCX.Beckhoff_CUxxxx.Beckhoff_CUxxxxEK1122.A_0001_CU1123_0000_0016.A_0002_CU1123_0010_0016.A_0003_CU1124_0000_0016.A_0004_CU1128_0000_0000.A_0005_CU1128_0000_0001.A_0006_CU1128_0000_0002.A_0011_CU2508_0000_0017.EPM_Inputs_Channel_8.Dropped_frames_tx <-> EPM Inputs Channel 8/Dropped frames tx
//     PlcTask Inputs/GVL_iXlinker.EtherCAT_Master_BKCUCX.Beckhoff_CUxxxx.Beckhoff_CUxxxxEK1122.A_0001_CU1123_0000_0016.A_0002_CU1123_0010_0016.A_0003_CU1124_0000_0016.A_0004_CU1128_0000_0000.A_0005_CU1128_0000_0001.A_0006_CU1128_0000_0002.A_0011_CU2508_0000_0017.EPM_Inputs_Channel_9.Dropped_frames_tx <-> EPM Inputs Channel 9/Dropped frames tx
//     PlcTask Inputs/GVL_iXlinker.EtherCAT_Master_BKCUCX.Beckhoff_CUxxxx.Beckhoff_CUxxxxEK1122.A_0001_CU1123_0000_0016.A_0002_CU1123_0010_0016.A_0003_CU1124_0000_0016.A_0004_CU1128_0000_0000.A_0005_CU1128_0000_0001.A_0006_CU1128_0000_0002.A_0011_CU2508_0000_0017.EPM_Inputs_Channel_10.Dropped_frames_tx <-> EPM Inputs Channel 10/Dropped frames tx
//     PlcTask Inputs/GVL_iXlinker.EtherCAT_Master_BKCUCX.Beckhoff_CUxxxx.Beckhoff_CUxxxxEK1122.A_0001_CU1123_0000_0016.A_0002_CU1123_0010_0016.A_0003_CU1124_0000_0016.A_0004_CU1128_0000_0000.A_0005_CU1128_0000_0001.A_0006_CU1128_0000_0002.A_0011_CU2508_0000_0017.WcState.WcState <-> WcState/WcState
//     PlcTask Inputs/GVL_iXlinker.EtherCAT_Master_BKCUCX.Beckhoff_CUxxxx.Beckhoff_CUxxxxEK1122.A_0001_CU1123_0000_0016.A_0002_CU1123_0010_0016.A_0003_CU1124_0000_0016.A_0004_CU1128_0000_0000.A_0005_CU1128_0000_0001.A_0006_CU1128_0000_0002.A_0011_CU2508_0000_0017.WcState.InputToggle <-> WcState/InputToggle
//     PlcTask Inputs/GVL_iXlinker.EtherCAT_Master_BKCUCX.Beckhoff_CUxxxx.Beckhoff_CUxxxxEK1122.A_0001_CU1123_0000_0016.A_0002_CU1123_0010_0016.A_0003_CU1124_0000_0016.A_0004_CU1128_0000_0000.A_0005_CU1128_0000_0001.A_0006_CU1128_0000_0002.A_0011_CU2508_0000_0017.InfoData.AdsAddr <-> InfoData/AdsAddr
//     PlcTask Inputs/GVL_iXlinker.EtherCAT_Master_BKCUCX.Beckhoff_CUxxxx.Beckhoff_CUxxxxEK1122.A_0001_CU1123_0000_0016.A_0002_CU1123_0010_0016.A_0003_CU1124_0000_0016.A_0004_CU1128_0000_0000.A_0005_CU1128_0000_0001.A_0006_CU1128_0000_0002.A_0011_CU2508_0000_0017.InfoData.State <-> InfoData/State
//   PLC/PLC Instance <-> EtherCAT Master BKCUCX/Beckhoff CUxxxx/Beckhoff CUxxxxEK1122/A_0001(CU1123-0000-0016)/A_0002(CU1123-0010-0016)/A_0003(CU1124-0000-0016)/A_0004(CU1128-0000-0000)/A_0005(CU1128-0000-0001)/A_0006(CU1128-0000-0002)/A_0012(CU2508-0000-0018)
//     PlcTask Inputs/GVL_iXlinker.EtherCAT_Master_BKCUCX.Beckhoff_CUxxxx.Beckhoff_CUxxxxEK1122.A_0001_CU1123_0000_0016.A_0002_CU1123_0010_0016.A_0003_CU1124_0000_0016.A_0004_CU1128_0000_0000.A_0005_CU1128_0000_0001.A_0006_CU1128_0000_0002.A_0012_CU2508_0000_0018.EPM_Inputs_Channel_1.Dropped_frames_rx <-> EPM Inputs Channel 1/Dropped frames rx
//     PlcTask Inputs/GVL_iXlinker.EtherCAT_Master_BKCUCX.Beckhoff_CUxxxx.Beckhoff_CUxxxxEK1122.A_0001_CU1123_0000_0016.A_0002_CU1123_0010_0016.A_0003_CU1124_0000_0016.A_0004_CU1128_0000_0000.A_0005_CU1128_0000_0001.A_0006_CU1128_0000_0002.A_0012_CU2508_0000_0018.EPM_Inputs_Channel_2.Dropped_frames_rx <-> EPM Inputs Channel 2/Dropped frames rx
//     PlcTask Inputs/GVL_iXlinker.EtherCAT_Master_BKCUCX.Beckhoff_CUxxxx.Beckhoff_CUxxxxEK1122.A_0001_CU1123_0000_0016.A_0002_CU1123_0010_0016.A_0003_CU1124_0000_0016.A_0004_CU1128_0000_0000.A_0005_CU1128_0000_0001.A_0006_CU1128_0000_0002.A_0012_CU2508_0000_0018.EPM_Inputs_Channel_3.Dropped_frames_rx <-> EPM Inputs Channel 3/Dropped frames rx
//     PlcTask Inputs/GVL_iXlinker.EtherCAT_Master_BKCUCX.Beckhoff_CUxxxx.Beckhoff_CUxxxxEK1122.A_0001_CU1123_0000_0016.A_0002_CU1123_0010_0016.A_0003_CU1124_0000_0016.A_0004_CU1128_0000_0000.A_0005_CU1128_0000_0001.A_0006_CU1128_0000_0002.A_0012_CU2508_0000_0018.EPM_Inputs_Channel_4.Dropped_frames_rx <-> EPM Inputs Channel 4/Dropped frames rx
//     PlcTask Inputs/GVL_iXlinker.EtherCAT_Master_BKCUCX.Beckhoff_CUxxxx.Beckhoff_CUxxxxEK1122.A_0001_CU1123_0000_0016.A_0002_CU1123_0010_0016.A_0003_CU1124_0000_0016.A_0004_CU1128_0000_0000.A_0005_CU1128_0000_0001.A_0006_CU1128_0000_0002.A_0012_CU2508_0000_0018.EPM_Inputs_Channel_5.Dropped_frames_rx <-> EPM Inputs Channel 5/Dropped frames rx
//     PlcTask Inputs/GVL_iXlinker.EtherCAT_Master_BKCUCX.Beckhoff_CUxxxx.Beckhoff_CUxxxxEK1122.A_0001_CU1123_0000_0016.A_0002_CU1123_0010_0016.A_0003_CU1124_0000_0016.A_0004_CU1128_0000_0000.A_0005_CU1128_0000_0001.A_0006_CU1128_0000_0002.A_0012_CU2508_0000_0018.EPM_Inputs_Channel_6.Dropped_frames_rx <-> EPM Inputs Channel 6/Dropped frames rx
//     PlcTask Inputs/GVL_iXlinker.EtherCAT_Master_BKCUCX.Beckhoff_CUxxxx.Beckhoff_CUxxxxEK1122.A_0001_CU1123_0000_0016.A_0002_CU1123_0010_0016.A_0003_CU1124_0000_0016.A_0004_CU1128_0000_0000.A_0005_CU1128_0000_0001.A_0006_CU1128_0000_0002.A_0012_CU2508_0000_0018.EPM_Inputs_Channel_7.Dropped_frames_rx <-> EPM Inputs Channel 7/Dropped frames rx
//     PlcTask Inputs/GVL_iXlinker.EtherCAT_Master_BKCUCX.Beckhoff_CUxxxx.Beckhoff_CUxxxxEK1122.A_0001_CU1123_0000_0016.A_0002_CU1123_0010_0016.A_0003_CU1124_0000_0016.A_0004_CU1128_0000_0000.A_0005_CU1128_0000_0001.A_0006_CU1128_0000_0002.A_0012_CU2508_0000_0018.EPM_Inputs_Channel_8.Dropped_frames_rx <-> EPM Inputs Channel 8/Dropped frames rx
//     PlcTask Inputs/GVL_iXlinker.EtherCAT_Master_BKCUCX.Beckhoff_CUxxxx.Beckhoff_CUxxxxEK1122.A_0001_CU1123_0000_0016.A_0002_CU1123_0010_0016.A_0003_CU1124_0000_0016.A_0004_CU1128_0000_0000.A_0005_CU1128_0000_0001.A_0006_CU1128_0000_0002.A_0012_CU2508_0000_0018.EPM_Inputs_Channel_9.Dropped_frames_rx <-> EPM Inputs Channel 9/Dropped frames rx
//     PlcTask Inputs/GVL_iXlinker.EtherCAT_Master_BKCUCX.Beckhoff_CUxxxx.Beckhoff_CUxxxxEK1122.A_0001_CU1123_0000_0016.A_0002_CU1123_0010_0016.A_0003_CU1124_0000_0016.A_0004_CU1128_0000_0000.A_0005_CU1128_0000_0001.A_0006_CU1128_0000_0002.A_0012_CU2508_0000_0018.EPM_Inputs_Channel_10.Dropped_frames_rx <-> EPM Inputs Channel 10/Dropped frames rx
//     PlcTask Inputs/GVL_iXlinker.EtherCAT_Master_BKCUCX.Beckhoff_CUxxxx.Beckhoff_CUxxxxEK1122.A_0001_CU1123_0000_0016.A_0002_CU1123_0010_0016.A_0003_CU1124_0000_0016.A_0004_CU1128_0000_0000.A_0005_CU1128_0000_0001.A_0006_CU1128_0000_0002.A_0012_CU2508_0000_0018.EPM_Inputs_Channel_1.Dropped_frames_tx <-> EPM Inputs Channel 1/Dropped frames tx
//     PlcTask Inputs/GVL_iXlinker.EtherCAT_Master_BKCUCX.Beckhoff_CUxxxx.Beckhoff_CUxxxxEK1122.A_0001_CU1123_0000_0016.A_0002_CU1123_0010_0016.A_0003_CU1124_0000_0016.A_0004_CU1128_0000_0000.A_0005_CU1128_0000_0001.A_0006_CU1128_0000_0002.A_0012_CU2508_0000_0018.EPM_Inputs_Channel_2.Dropped_frames_tx <-> EPM Inputs Channel 2/Dropped frames tx
//     PlcTask Inputs/GVL_iXlinker.EtherCAT_Master_BKCUCX.Beckhoff_CUxxxx.Beckhoff_CUxxxxEK1122.A_0001_CU1123_0000_0016.A_0002_CU1123_0010_0016.A_0003_CU1124_0000_0016.A_0004_CU1128_0000_0000.A_0005_CU1128_0000_0001.A_0006_CU1128_0000_0002.A_0012_CU2508_0000_0018.EPM_Inputs_Channel_3.Dropped_frames_tx <-> EPM Inputs Channel 3/Dropped frames tx
//     PlcTask Inputs/GVL_iXlinker.EtherCAT_Master_BKCUCX.Beckhoff_CUxxxx.Beckhoff_CUxxxxEK1122.A_0001_CU1123_0000_0016.A_0002_CU1123_0010_0016.A_0003_CU1124_0000_0016.A_0004_CU1128_0000_0000.A_0005_CU1128_0000_0001.A_0006_CU1128_0000_0002.A_0012_CU2508_0000_0018.EPM_Inputs_Channel_4.Dropped_frames_tx <-> EPM Inputs Channel 4/Dropped frames tx
//     PlcTask Inputs/GVL_iXlinker.EtherCAT_Master_BKCUCX.Beckhoff_CUxxxx.Beckhoff_CUxxxxEK1122.A_0001_CU1123_0000_0016.A_0002_CU1123_0010_0016.A_0003_CU1124_0000_0016.A_0004_CU1128_0000_0000.A_0005_CU1128_0000_0001.A_0006_CU1128_0000_0002.A_0012_CU2508_0000_0018.EPM_Inputs_Channel_5.Dropped_frames_tx <-> EPM Inputs Channel 5/Dropped frames tx
//     PlcTask Inputs/GVL_iXlinker.EtherCAT_Master_BKCUCX.Beckhoff_CUxxxx.Beckhoff_CUxxxxEK1122.A_0001_CU1123_0000_0016.A_0002_CU1123_0010_0016.A_0003_CU1124_0000_0016.A_0004_CU1128_0000_0000.A_0005_CU1128_0000_0001.A_0006_CU1128_0000_0002.A_0012_CU2508_0000_0018.EPM_Inputs_Channel_6.Dropped_frames_tx <-> EPM Inputs Channel 6/Dropped frames tx
//     PlcTask Inputs/GVL_iXlinker.EtherCAT_Master_BKCUCX.Beckhoff_CUxxxx.Beckhoff_CUxxxxEK1122.A_0001_CU1123_0000_0016.A_0002_CU1123_0010_0016.A_0003_CU1124_0000_0016.A_0004_CU1128_0000_0000.A_0005_CU1128_0000_0001.A_0006_CU1128_0000_0002.A_0012_CU2508_0000_0018.EPM_Inputs_Channel_7.Dropped_frames_tx <-> EPM Inputs Channel 7/Dropped frames tx
//     PlcTask Inputs/GVL_iXlinker.EtherCAT_Master_BKCUCX.Beckhoff_CUxxxx.Beckhoff_CUxxxxEK1122.A_0001_CU1123_0000_0016.A_0002_CU1123_0010_0016.A_0003_CU1124_0000_0016.A_0004_CU1128_0000_0000.A_0005_CU1128_0000_0001.A_0006_CU1128_0000_0002.A_0012_CU2508_0000_0018.EPM_Inputs_Channel_8.Dropped_frames_tx <-> EPM Inputs Channel 8/Dropped frames tx
//     PlcTask Inputs/GVL_iXlinker.EtherCAT_Master_BKCUCX.Beckhoff_CUxxxx.Beckhoff_CUxxxxEK1122.A_0001_CU1123_0000_0016.A_0002_CU1123_0010_0016.A_0003_CU1124_0000_0016.A_0004_CU1128_0000_0000.A_0005_CU1128_0000_0001.A_0006_CU1128_0000_0002.A_0012_CU2508_0000_0018.EPM_Inputs_Channel_9.Dropped_frames_tx <-> EPM Inputs Channel 9/Dropped frames tx
//     PlcTask Inputs/GVL_iXlinker.EtherCAT_Master_BKCUCX.Beckhoff_CUxxxx.Beckhoff_CUxxxxEK1122.A_0001_CU1123_0000_0016.A_0002_CU1123_0010_0016.A_0003_CU1124_0000_0016.A_0004_CU1128_0000_0000.A_0005_CU1128_0000_0001.A_0006_CU1128_0000_0002.A_0012_CU2508_0000_0018.EPM_Inputs_Channel_10.Dropped_frames_tx <-> EPM Inputs Channel 10/Dropped frames tx
//     PlcTask Inputs/GVL_iXlinker.EtherCAT_Master_BKCUCX.Beckhoff_CUxxxx.Beckhoff_CUxxxxEK1122.A_0001_CU1123_0000_0016.A_0002_CU1123_0010_0016.A_0003_CU1124_0000_0016.A_0004_CU1128_0000_0000.A_0005_CU1128_0000_0001.A_0006_CU1128_0000_0002.A_0012_CU2508_0000_0018.WcState.WcState <-> WcState/WcState
//     PlcTask Inputs/GVL_iXlinker.EtherCAT_Master_BKCUCX.Beckhoff_CUxxxx.Beckhoff_CUxxxxEK1122.A_0001_CU1123_0000_0016.A_0002_CU1123_0010_0016.A_0003_CU1124_0000_0016.A_0004_CU1128_0000_0000.A_0005_CU1128_0000_0001.A_0006_CU1128_0000_0002.A_0012_CU2508_0000_0018.WcState.InputToggle <-> WcState/InputToggle
//     PlcTask Inputs/GVL_iXlinker.EtherCAT_Master_BKCUCX.Beckhoff_CUxxxx.Beckhoff_CUxxxxEK1122.A_0001_CU1123_0000_0016.A_0002_CU1123_0010_0016.A_0003_CU1124_0000_0016.A_0004_CU1128_0000_0000.A_0005_CU1128_0000_0001.A_0006_CU1128_0000_0002.A_0012_CU2508_0000_0018.InfoData.AdsAddr <-> InfoData/AdsAddr
//     PlcTask Inputs/GVL_iXlinker.EtherCAT_Master_BKCUCX.Beckhoff_CUxxxx.Beckhoff_CUxxxxEK1122.A_0001_CU1123_0000_0016.A_0002_CU1123_0010_0016.A_0003_CU1124_0000_0016.A_0004_CU1128_0000_0000.A_0005_CU1128_0000_0001.A_0006_CU1128_0000_0002.A_0012_CU2508_0000_0018.InfoData.State <-> InfoData/State
//   PLC/PLC Instance <-> EtherCAT Master BKCUCX/Beckhoff CUxxxx/Beckhoff CUxxxxEK1122/A_0001(CU1123-0000-0016)/A_0002(CU1123-0010-0016)/A_0003(CU1124-0000-0016)/A_0004(CU1128-0000-0000)/A_0005(CU1128-0000-0001)/A_0006(CU1128-0000-0002)/A_0013(CU2508-0000-0019)
//     PlcTask Inputs/GVL_iXlinker.EtherCAT_Master_BKCUCX.Beckhoff_CUxxxx.Beckhoff_CUxxxxEK1122.A_0001_CU1123_0000_0016.A_0002_CU1123_0010_0016.A_0003_CU1124_0000_0016.A_0004_CU1128_0000_0000.A_0005_CU1128_0000_0001.A_0006_CU1128_0000_0002.A_0013_CU2508_0000_0019.EPM_Inputs_Channel_1.Dropped_frames_rx <-> EPM Inputs Channel 1/Dropped frames rx
//     PlcTask Inputs/GVL_iXlinker.EtherCAT_Master_BKCUCX.Beckhoff_CUxxxx.Beckhoff_CUxxxxEK1122.A_0001_CU1123_0000_0016.A_0002_CU1123_0010_0016.A_0003_CU1124_0000_0016.A_0004_CU1128_0000_0000.A_0005_CU1128_0000_0001.A_0006_CU1128_0000_0002.A_0013_CU2508_0000_0019.EPM_Inputs_Channel_2.Dropped_frames_rx <-> EPM Inputs Channel 2/Dropped frames rx
//     PlcTask Inputs/GVL_iXlinker.EtherCAT_Master_BKCUCX.Beckhoff_CUxxxx.Beckhoff_CUxxxxEK1122.A_0001_CU1123_0000_0016.A_0002_CU1123_0010_0016.A_0003_CU1124_0000_0016.A_0004_CU1128_0000_0000.A_0005_CU1128_0000_0001.A_0006_CU1128_0000_0002.A_0013_CU2508_0000_0019.EPM_Inputs_Channel_3.Dropped_frames_rx <-> EPM Inputs Channel 3/Dropped frames rx
//     PlcTask Inputs/GVL_iXlinker.EtherCAT_Master_BKCUCX.Beckhoff_CUxxxx.Beckhoff_CUxxxxEK1122.A_0001_CU1123_0000_0016.A_0002_CU1123_0010_0016.A_0003_CU1124_0000_0016.A_0004_CU1128_0000_0000.A_0005_CU1128_0000_0001.A_0006_CU1128_0000_0002.A_0013_CU2508_0000_0019.EPM_Inputs_Channel_4.Dropped_frames_rx <-> EPM Inputs Channel 4/Dropped frames rx
//     PlcTask Inputs/GVL_iXlinker.EtherCAT_Master_BKCUCX.Beckhoff_CUxxxx.Beckhoff_CUxxxxEK1122.A_0001_CU1123_0000_0016.A_0002_CU1123_0010_0016.A_0003_CU1124_0000_0016.A_0004_CU1128_0000_0000.A_0005_CU1128_0000_0001.A_0006_CU1128_0000_0002.A_0013_CU2508_0000_0019.EPM_Inputs_Channel_5.Dropped_frames_rx <-> EPM Inputs Channel 5/Dropped frames rx
//     PlcTask Inputs/GVL_iXlinker.EtherCAT_Master_BKCUCX.Beckhoff_CUxxxx.Beckhoff_CUxxxxEK1122.A_0001_CU1123_0000_0016.A_0002_CU1123_0010_0016.A_0003_CU1124_0000_0016.A_0004_CU1128_0000_0000.A_0005_CU1128_0000_0001.A_0006_CU1128_0000_0002.A_0013_CU2508_0000_0019.EPM_Inputs_Channel_6.Dropped_frames_rx <-> EPM Inputs Channel 6/Dropped frames rx
//     PlcTask Inputs/GVL_iXlinker.EtherCAT_Master_BKCUCX.Beckhoff_CUxxxx.Beckhoff_CUxxxxEK1122.A_0001_CU1123_0000_0016.A_0002_CU1123_0010_0016.A_0003_CU1124_0000_0016.A_0004_CU1128_0000_0000.A_0005_CU1128_0000_0001.A_0006_CU1128_0000_0002.A_0013_CU2508_0000_0019.EPM_Inputs_Channel_7.Dropped_frames_rx <-> EPM Inputs Channel 7/Dropped frames rx
//     PlcTask Inputs/GVL_iXlinker.EtherCAT_Master_BKCUCX.Beckhoff_CUxxxx.Beckhoff_CUxxxxEK1122.A_0001_CU1123_0000_0016.A_0002_CU1123_0010_0016.A_0003_CU1124_0000_0016.A_0004_CU1128_0000_0000.A_0005_CU1128_0000_0001.A_0006_CU1128_0000_0002.A_0013_CU2508_0000_0019.EPM_Inputs_Channel_8.Dropped_frames_rx <-> EPM Inputs Channel 8/Dropped frames rx
//     PlcTask Inputs/GVL_iXlinker.EtherCAT_Master_BKCUCX.Beckhoff_CUxxxx.Beckhoff_CUxxxxEK1122.A_0001_CU1123_0000_0016.A_0002_CU1123_0010_0016.A_0003_CU1124_0000_0016.A_0004_CU1128_0000_0000.A_0005_CU1128_0000_0001.A_0006_CU1128_0000_0002.A_0013_CU2508_0000_0019.EPM_Inputs_Channel_9.Dropped_frames_rx <-> EPM Inputs Channel 9/Dropped frames rx
//     PlcTask Inputs/GVL_iXlinker.EtherCAT_Master_BKCUCX.Beckhoff_CUxxxx.Beckhoff_CUxxxxEK1122.A_0001_CU1123_0000_0016.A_0002_CU1123_0010_0016.A_0003_CU1124_0000_0016.A_0004_CU1128_0000_0000.A_0005_CU1128_0000_0001.A_0006_CU1128_0000_0002.A_0013_CU2508_0000_0019.EPM_Inputs_Channel_10.Dropped_frames_rx <-> EPM Inputs Channel 10/Dropped frames rx
